LIN {X 0,Y 251.321,Z 689.744,A -85,B 0,C 180,E1 12849.752,E2 12849.752} C_VEL
LIN {X 0,Y 252.942,Z 676.86,A -85,B 0,C 180,E1 12846.595,E2 12846.595} C_VEL
LIN {X 0,Y 255.041,Z 662.352,A -85,B 0,C 180,E1 12843.706,E2 12843.706} C_VEL
LIN {X 0,Y 257.379,Z 646.816,A -85,B 0,C 180,E1 12841.205,E2 12841.205} C_VEL
LIN {X 0,Y 259.787,Z 630.262,A -85,B 0,C 180,E1 12839.084,E2 12839.084} C_VEL
LIN {X 0,Y 262.1,Z 612.775,A -85,B 0,C 180,E1 12837.333,E2 12837.333} C_VEL
LIN {X 0,Y 264.21,Z 594.401,A -85,B 0,C 180,E1 12835.941,E2 12835.941} C_VEL
LIN {X 0,Y 265.742,Z 575.64,A -85,B 0,C 180,E1 12834.93,E2 12834.93} C_VEL
LIN {X 0,Y 274.022,Z 424.566,A -85,B 0,C 180,E1 12829.575,E2 12829.575} C_VEL
LIN {X 0,Y 272.391,Z 392.722,A -85,B 0,C 180,E1 12828.155,E2 12828.155} C_VEL
LIN {X 0,Y 272.465,Z 390.527,A -85,B 0,C 180,E1 12828.028,E2 12828.028} C_VEL
LIN {X 0,Y 273.095,Z 387.473,A -85,B 0,C 180,E1 12827.542,E2 12827.542} C_VEL
LIN {X 0,Y 266.657,Z 366.923,A -85,B 0,C 180,E1 12823.018,E2 12823.018} C_VEL
LIN {X 0,Y 260.852,Z 349.171,A -85,B 0,C 180,E1 12818.67,E2 12818.67} C_VEL
LIN {X 0,Y 255.343,Z 333.14,A -85,B 0,C 180,E1 12814.327,E2 12814.327} C_VEL
LIN {X 0,Y 250.605,Z 319.583,A -85,B 0,C 180,E1 12810.252,E2 12810.252} C_VEL
LIN {X 0,Y 250.621,Z 319.582,A -85,B 0,C 180,E1 12805.526,E2 12805.526} C_VEL
LIN {X 0,Y 250.603,Z 319.579,A -85,B 0,C 180,E1 12800.558,E2 12800.558} C_VEL
LIN {X 0,Y 250.63,Z 319.58,A -85,B 0,C 180,E1 12795.506,E2 12795.506} C_VEL
LIN {X 0,Y 250.608,Z 319.58,A -85,B 0,C 180,E1 12790.346,E2 12790.346} C_VEL
LIN {X 0,Y 250.626,Z 319.579,A -85,B 0,C 180,E1 12785.497,E2 12785.497} C_VEL
LIN {X 0,Y 250.606,Z 319.58,A -85,B 0,C 180,E1 12780.46,E2 12780.46} C_VEL
LIN {X 0,Y 250.625,Z 319.576,A -85,B 0,C 180,E1 12775.427,E2 12775.427} C_VEL
LIN {X 0,Y 250.607,Z 319.572,A -85,B 0,C 180,E1 12770.589,E2 12770.589} C_VEL
LIN {X 0,Y 250.645,Z 319.578,A -85,B 0,C 180,E1 12765.448,E2 12765.448} C_VEL
LIN {X 0,Y 250.613,Z 319.565,A -85,B 0,C 180,E1 12760.309,E2 12760.309} C_VEL
LIN {X 0,Y 250.635,Z 319.578,A -85,B 0,C 180,E1 12755.44,E2 12755.44} C_VEL
LIN {X 0,Y 250.614,Z 319.559,A -85,B 0,C 180,E1 12750.425,E2 12750.425} C_VEL
LIN {X 0,Y 250.636,Z 319.579,A -85,B 0,C 180,E1 12745.5,E2 12745.5} C_VEL
LIN {X 0,Y 250.619,Z 319.565,A -85,B 0,C 180,E1 12740.634,E2 12740.634} C_VEL
LIN {X 0,Y 250.636,Z 319.572,A -85,B 0,C 180,E1 12735.565,E2 12735.565} C_VEL
LIN {X 0,Y 250.619,Z 319.573,A -85,B 0,C 180,E1 12730.562,E2 12730.562} C_VEL
LIN {X 0,Y 250.633,Z 319.56,A -85,B 0,C 180,E1 12725.536,E2 12725.536} C_VEL
LIN {X 0,Y 250.627,Z 319.577,A -85,B 0,C 180,E1 12720.705,E2 12720.705} C_VEL
LIN {X 0,Y 250.636,Z 319.561,A -85,B 0,C 180,E1 12715.644,E2 12715.644} C_VEL
LIN {X 0,Y 250.634,Z 319.574,A -85,B 0,C 180,E1 12710.794,E2 12710.794} C_VEL
LIN {X 0,Y 250.635,Z 319.571,A -85,B 0,C 180,E1 12705.738,E2 12705.738} C_VEL
LIN {X 0,Y 250.635,Z 319.574,A -85,B 0,C 180,E1 12700.805,E2 12700.805} C_VEL
LIN {X 0,Y 250.634,Z 319.573,A -85,B 0,C 180,E1 12695.722,E2 12695.722} C_VEL
LIN {X 0,Y 250.638,Z 319.575,A -85,B 0,C 180,E1 12690.684,E2 12690.684} C_VEL
LIN {X 0,Y 250.636,Z 319.567,A -85,B 0,C 180,E1 12685.651,E2 12685.651} C_VEL
LIN {X 0,Y 250.645,Z 319.572,A -85,B 0,C 180,E1 12680.817,E2 12680.817} C_VEL
LIN {X 0,Y 250.639,Z 319.578,A -85,B 0,C 180,E1 12675.679,E2 12675.679} C_VEL
LIN {X 0,Y 250.651,Z 319.575,A -85,B 0,C 180,E1 12670.905,E2 12670.905} C_VEL
LIN {X 0,Y 250.639,Z 319.578,A -85,B 0,C 180,E1 12665.737,E2 12665.737} C_VEL
LIN {X 0,Y 250.66,Z 319.574,A -85,B 0,C 180,E1 12660.867,E2 12660.867} C_VEL
LIN {X 0,Y 250.639,Z 319.575,A -85,B 0,C 180,E1 12655.77,E2 12655.77} C_VEL
LIN {X 0,Y 250.691,Z 319.79,A -85,B 0,C 180,E1 12651.229,E2 12651.229} C_VEL
LIN {X 0,Y 255.331,Z 334.84,A -85,B 0,C 180,E1 12646.417,E2 12646.417} C_VEL
LIN {X 0,Y 259.574,Z 349.98,A -85,B 0,C 180,E1 12641.974,E2 12641.974} C_VEL
LIN {X 0,Y 263.572,Z 365.649,A -85,B 0,C 180,E1 12637.706,E2 12637.706} C_VEL
LIN {X 0,Y 265.522,Z 374.511,A -85,B 0,C 180,E1 12635.439,E2 12635.439} C_VEL
LIN {X 0,Y 260.741,Z 400.55,A -85,B 0,C 180,E1 12630.016,E2 12630.016} C_VEL
LIN {X 0,Y 264.226,Z 442.101,A -85,B 0,C 180,E1 12627.745,E2 12627.745} C_VEL
LIN {X 0,Y 258.452,Z 538.649,A -85,B 0,C 180,E1 12623.423,E2 12623.423} C_VEL
LIN {X 0,Y 257.316,Z 556.591,A -85,B 0,C 180,E1 12622.208,E2 12622.208} C_VEL
LIN {X 0,Y 256.049,Z 573.142,A -85,B 0,C 180,E1 12620.691,E2 12620.691} C_VEL
LIN {X 0,Y 254.557,Z 590.125,A -85,B 0,C 180,E1 12618.666,E2 12618.666} C_VEL
LIN {X 0,Y 253.14,Z 605.769,A -85,B 0,C 180,E1 12616.283,E2 12616.283} C_VEL
LIN {X 0,Y 251.879,Z 620.01,A -85,B 0,C 180,E1 12613.541,E2 12613.541} C_VEL
LIN {X 0,Y 250.936,Z 632.25,A -85,B 0,C 180,E1 12610.558,E2 12610.558} C_VEL
LIN {X 0,Y 250.407,Z 642.044,A -85,B 0,C 180,E1 12607.568,E2 12607.568} C_VEL
LIN {X 0,Y 250.249,Z 650.429,A -85,B 0,C 180,E1 12604.35,E2 12604.35} C_VEL
LIN {X 0,Y 250.336,Z 654.067,A -85,B 0,C 180,E1 12602.603,E2 12602.603} C_VEL
LIN {X 0,Y 249.534,Z 657.084,A -85,B 0,C 180,E1 12600.972,E2 12600.972} C_VEL
LIN {X 0,Y 245.629,Z 662.003,A -85,B 0,C 180,E1 12597.788,E2 12597.788} C_VEL
LIN {X 0,Y 244.226,Z 664.446,A -85,B 0,C 180,E1 12595.666,E2 12595.666} C_VEL
LIN {X 0,Y 244.363,Z 665.1,A -85,B 0,C 180,E1 12594.901,E2 12594.901} C_VEL
LIN {X 0,Y 246.382,Z 667.107,A -85,B 0,C 180,E1 12591.361,E2 12591.361} C_VEL
LIN {X 0,Y 249.308,Z 667.226,A -85,B 0,C 180,E1 12587.725,E2 12587.725} C_VEL
LIN {X 0,Y 253.145,Z 665.497,A -85,B 0,C 180,E1 12584.182,E2 12584.182} C_VEL
LIN {X 0,Y 257.872,Z 661.812,A -85,B 0,C 180,E1 12580.754,E2 12580.754} C_VEL
LIN {X 0,Y 263.52,Z 656.236,A -85,B 0,C 180,E1 12577.464,E2 12577.464} C_VEL
LIN {X 0,Y 270.049,Z 648.574,A -85,B 0,C 180,E1 12574.327,E2 12574.327} C_VEL
LIN {X 0,Y 276.967,Z 639.386,A -85,B 0,C 180,E1 12571.539,E2 12571.539} C_VEL
LIN {X 0,Y 284.686,Z 628.026,A -85,B 0,C 180,E1 12568.914,E2 12568.914} C_VEL
LIN {X 0,Y 292.903,Z 614.48,A -85,B 0,C 180,E1 12566.541,E2 12566.541} C_VEL
LIN {X 0,Y 300.548,Z 600.238,A -85,B 0,C 180,E1 12564.627,E2 12564.627} C_VEL
LIN {X 0,Y 307.744,Z 584.985,A -85,B 0,C 180,E1 12563.051,E2 12563.051} C_VEL
LIN {X 0,Y 314.232,Z 568.47,A -85,B 0,C 180,E1 12561.763,E2 12561.763} C_VEL
LIN {X 0,Y 319.672,Z 551.343,A -85,B 0,C 180,E1 12560.771,E2 12560.771} C_VEL
LIN {X 0,Y 325.594,Z 530.519,A -85,B 0,C 180,E1 12559.792,E2 12559.792} C_VEL
LIN {X 0,Y 315.19,Z 568.695,A -85,B 0,C 180,E1 12558.338,E2 12558.338} C_VEL
LIN {X 0,Y 307.601,Z 590.208,A -85,B 0,C 180,E1 12557.276,E2 12557.276} C_VEL
LIN {X 0,Y 299.978,Z 608.25,A -85,B 0,C 180,E1 12556.052,E2 12556.052} C_VEL
LIN {X 0,Y 291.443,Z 626.077,A -85,B 0,C 180,E1 12554.418,E2 12554.418} C_VEL
LIN {X 0,Y 282.982,Z 642.204,A -85,B 0,C 180,E1 12552.445,E2 12552.445} C_VEL
LIN {X 0,Y 274.169,Z 657.891,A -85,B 0,C 180,E1 12549.932,E2 12549.932} C_VEL
LIN {X 0,Y 265.896,Z 672.135,A -85,B 0,C 180,E1 12546.99,E2 12546.99} C_VEL
LIN {X 0,Y 258.373,Z 684.983,A -85,B 0,C 180,E1 12543.601,E2 12543.601} C_VEL
LIN {X 0,Y 251.862,Z 696.369,A -85,B 0,C 180,E1 12539.753,E2 12539.753} C_VEL
LIN {X 0,Y 246.671,Z 706.308,A -85,B 0,C 180,E1 12535.448,E2 12535.448} C_VEL
LIN {X 0,Y 243.156,Z 714.309,A -85,B 0,C 180,E1 12530.964,E2 12530.964} C_VEL
LIN {X 0,Y 241.284,Z 720.475,A -85,B 0,C 180,E1 12526.369,E2 12526.369} C_VEL
LIN {X 0,Y 240.873,Z 724.951,A -85,B 0,C 180,E1 12521.574,E2 12521.574} C_VEL
LIN {X 0,Y 241.603,Z 727.321,A -85,B 0,C 180,E1 12517.134,E2 12517.134} C_VEL
LIN {X 0,Y 242.656,Z 727.848,A -85,B 0,C 180,E1 12513.309,E2 12513.309} C_VEL
LIN {X 0,Y 243.307,Z 726.953,A -85,B 0,C 180,E1 12510.002,E2 12510.002} C_VEL
LIN {X 0,Y 243.197,Z 724.887,A -85,B 0,C 180,E1 12506.938,E2 12506.938} C_VEL
LIN {X 0,Y 242.612,Z 720.804,A -85,B 0,C 180,E1 12503.34,E2 12503.34} C_VEL
LIN {X 0,Y 242.105,Z 715.047,A -85,B 0,C 180,E1 12499.773,E2 12499.773} C_VEL
LIN {X 0,Y 242.009,Z 707.373,A -85,B 0,C 180,E1 12496.137,E2 12496.137} C_VEL
LIN {X 0,Y 242.521,Z 697.577,A -85,B 0,C 180,E1 12492.487,E2 12492.487} C_VEL
LIN {X 0,Y 243.672,Z 686.258,A -85,B 0,C 180,E1 12489.087,E2 12489.087} C_VEL
LIN {X 0,Y 245.402,Z 673.121,A -85,B 0,C 180,E1 12485.881,E2 12485.881} C_VEL
LIN {X 0,Y 247.487,Z 659.126,A -85,B 0,C 180,E1 12483.099,E2 12483.099} C_VEL
LIN {X 0,Y 249.818,Z 643.804,A -85,B 0,C 180,E1 12480.643,E2 12480.643} C_VEL
LIN {X 0,Y 252.319,Z 626.753,A -85,B 0,C 180,E1 12478.464,E2 12478.464} C_VEL
LIN {X 0,Y 254.732,Z 608.718,A -85,B 0,C 180,E1 12476.668,E2 12476.668} C_VEL
LIN {X 0,Y 256.805,Z 590.184,A -85,B 0,C 180,E1 12475.305,E2 12475.305} C_VEL
LIN {X 0,Y 258.241,Z 570.947,A -85,B 0,C 180,E1 12474.319,E2 12474.319} C_VEL
LIN {X 0,Y 266.563,Z 425.162,A -85,B 0,C 180,E1 12468.963,E2 12468.963} C_VEL
LIN {X 0,Y 265.03,Z 393.337,A -85,B 0,C 180,E1 12467.5,E2 12467.5} C_VEL
LIN {X 0,Y 265.123,Z 390.585,A -85,B 0,C 180,E1 12467.344,E2 12467.344} C_VEL
LIN {X 0,Y 265.183,Z 388.765,A -85,B 0,C 180,E1 12467.013,E2 12467.013} C_VEL
LIN {X 0,Y 258.711,Z 367.881,A -85,B 0,C 180,E1 12462.261,E2 12462.261} C_VEL
LIN {X 0,Y 252.668,Z 349.364,A -85,B 0,C 180,E1 12457.55,E2 12457.55} C_VEL
LIN {X 0,Y 246.993,Z 332.812,A -85,B 0,C 180,E1 12452.854,E2 12452.854} C_VEL
LIN {X 0,Y 242.667,Z 320.567,A -85,B 0,C 180,E1 12448.963,E2 12448.963} C_VEL
LIN {X 0,Y 242.684,Z 320.567,A -85,B 0,C 180,E1 12443.817,E2 12443.817} C_VEL
LIN {X 0,Y 242.666,Z 320.572,A -85,B 0,C 180,E1 12438.75,E2 12438.75} C_VEL
LIN {X 0,Y 242.686,Z 320.564,A -85,B 0,C 180,E1 12433.828,E2 12433.828} C_VEL
LIN {X 0,Y 242.665,Z 320.562,A -85,B 0,C 180,E1 12428.772,E2 12428.772} C_VEL
LIN {X 0,Y 242.681,Z 320.563,A -85,B 0,C 180,E1 12423.783,E2 12423.783} C_VEL
LIN {X 0,Y 242.671,Z 320.566,A -85,B 0,C 180,E1 12418.823,E2 12418.823} C_VEL
LIN {X 0,Y 242.696,Z 320.569,A -85,B 0,C 180,E1 12413.617,E2 12413.617} C_VEL
LIN {X 0,Y 242.671,Z 320.561,A -85,B 0,C 180,E1 12408.597,E2 12408.597} C_VEL
LIN {X 0,Y 242.695,Z 320.563,A -85,B 0,C 180,E1 12403.489,E2 12403.489} C_VEL
LIN {X 0,Y 242.676,Z 320.563,A -85,B 0,C 180,E1 12398.492,E2 12398.492} C_VEL
LIN {X 0,Y 242.698,Z 320.559,A -85,B 0,C 180,E1 12393.374,E2 12393.374} C_VEL
LIN {X 0,Y 242.678,Z 320.558,A -85,B 0,C 180,E1 12388.454,E2 12388.454} C_VEL
LIN {X 0,Y 242.696,Z 320.564,A -85,B 0,C 180,E1 12383.449,E2 12383.449} C_VEL
LIN {X 0,Y 242.679,Z 320.547,A -85,B 0,C 180,E1 12378.451,E2 12378.451} C_VEL
LIN {X 0,Y 242.7,Z 320.567,A -85,B 0,C 180,E1 12373.469,E2 12373.469} C_VEL
LIN {X 0,Y 242.681,Z 320.553,A -85,B 0,C 180,E1 12368.469,E2 12368.469} C_VEL
LIN {X 0,Y 242.702,Z 320.561,A -85,B 0,C 180,E1 12363.257,E2 12363.257} C_VEL
LIN {X 0,Y 242.688,Z 320.563,A -85,B 0,C 180,E1 12358.166,E2 12358.166} C_VEL
LIN {X 0,Y 242.703,Z 320.552,A -85,B 0,C 180,E1 12353.038,E2 12353.038} C_VEL
LIN {X 0,Y 242.696,Z 320.566,A -85,B 0,C 180,E1 12347.748,E2 12347.748} C_VEL
LIN {X 0,Y 242.698,Z 320.552,A -85,B 0,C 180,E1 12342.852,E2 12342.852} C_VEL
LIN {X 0,Y 242.702,Z 320.567,A -85,B 0,C 180,E1 12337.574,E2 12337.574} C_VEL
LIN {X 0,Y 242.693,Z 320.559,A -85,B 0,C 180,E1 12332.596,E2 12332.596} C_VEL
LIN {X 0,Y 242.704,Z 320.559,A -85,B 0,C 180,E1 12327.401,E2 12327.401} C_VEL
LIN {X 0,Y 242.694,Z 320.565,A -85,B 0,C 180,E1 12322.423,E2 12322.423} C_VEL
LIN {X 0,Y 242.708,Z 320.564,A -85,B 0,C 180,E1 12317.387,E2 12317.387} C_VEL
LIN {X 0,Y 242.7,Z 320.563,A -85,B 0,C 180,E1 12312.496,E2 12312.496} C_VEL
LIN {X 0,Y 242.724,Z 320.566,A -85,B 0,C 180,E1 12307.217,E2 12307.217} C_VEL
LIN {X 0,Y 242.701,Z 320.567,A -85,B 0,C 180,E1 12302.254,E2 12302.254} C_VEL
LIN {X 0,Y 242.718,Z 320.564,A -85,B 0,C 180,E1 12297.17,E2 12297.17} C_VEL
LIN {X 0,Y 242.708,Z 320.589,A -85,B 0,C 180,E1 12292.43,E2 12292.43} C_VEL
LIN {X 0,Y 247.265,Z 335.339,A -85,B 0,C 180,E1 12287.521,E2 12287.521} C_VEL
LIN {X 0,Y 251.505,Z 350.2,A -85,B 0,C 180,E1 12282.986,E2 12282.986} C_VEL
LIN {X 0,Y 255.595,Z 366.284,A -85,B 0,C 180,E1 12278.456,E2 12278.456} C_VEL
LIN {X 0,Y 257.838,Z 376.167,A -85,B 0,C 180,E1 12275.837,E2 12275.837} C_VEL
LIN {X 0,Y 253.208,Z 400.564,A -85,B 0,C 180,E1 12270.66,E2 12270.66} C_VEL
LIN {X 0,Y 256.409,Z 441.043,A -85,B 0,C 180,E1 12268.368,E2 12268.368} C_VEL
LIN {X 0,Y 256.416,Z 446.756,A -85,B 0,C 180,E1 12268.085,E2 12268.085} C_VEL
LIN {X 0,Y 250.616,Z 539.133,A -85,B 0,C 180,E1 12263.788,E2 12263.788} C_VEL
LIN {X 0,Y 249.42,Z 557.457,A -85,B 0,C 180,E1 12262.505,E2 12262.505} C_VEL
LIN {X 0,Y 248.079,Z 574.425,A -85,B 0,C 180,E1 12260.893,E2 12260.893} C_VEL
LIN {X 0,Y 246.636,Z 590.499,A -85,B 0,C 180,E1 12258.92,E2 12258.92} C_VEL
LIN {X 0,Y 245.114,Z 606.831,A -85,B 0,C 180,E1 12256.344,E2 12256.344} C_VEL
LIN {X 0,Y 243.838,Z 621.036,A -85,B 0,C 180,E1 12253.513,E2 12253.513} C_VEL
LIN {X 0,Y 242.86,Z 633.967,A -85,B 0,C 180,E1 12250.265,E2 12250.265} C_VEL
LIN {X 0,Y 242.364,Z 643.889,A -85,B 0,C 180,E1 12247.106,E2 12247.106} C_VEL
LIN {X 0,Y 242.273,Z 652.096,A -85,B 0,C 180,E1 12243.783,E2 12243.783} C_VEL
LIN {X 0,Y 242.676,Z 658.769,A -85,B 0,C 180,E1 12240.233,E2 12240.233} C_VEL
LIN {X 0,Y 243.628,Z 663.41,A -85,B 0,C 180,E1 12236.703,E2 12236.703} C_VEL
LIN {X 0,Y 244.363,Z 665.1,A -85,B 0,C 180,E1 12234.901,E2 12234.901} C_VEL
LIN {X 0,Y 244.306,Z 666.547,A -85,B 0,C 180,E1 12233.11,E2 12233.11} C_VEL
LIN {X 0,Y 241.997,Z 668.588,A -85,B 0,C 180,E1 12229.49,E2 12229.49} C_VEL
LIN {X 0,Y 241.842,Z 668.966,A -85,B 0,C 180,E1 12227.384,E2 12227.384} C_VEL
LIN {X 0,Y 242.405,Z 668.865,A -85,B 0,C 180,E1 12226.608,E2 12226.608} C_VEL
LIN {X 0,Y 246.611,Z 667.235,A -85,B 0,C 180,E1 12223.024,E2 12223.024} C_VEL
LIN {X 0,Y 252.134,Z 663.404,A -85,B 0,C 180,E1 12219.33,E2 12219.33} C_VEL
LIN {X 0,Y 258.313,Z 657.897,A -85,B 0,C 180,E1 12216.017,E2 12216.017} C_VEL
LIN {X 0,Y 265.885,Z 649.875,A -85,B 0,C 180,E1 12212.689,E2 12212.689} C_VEL
LIN {X 0,Y 273.919,Z 640.089,A -85,B 0,C 180,E1 12209.75,E2 12209.75} C_VEL
LIN {X 0,Y 281.716,Z 629.576,A -85,B 0,C 180,E1 12207.349,E2 12207.349} C_VEL
LIN {X 0,Y 290.837,Z 615.795,A -85,B 0,C 180,E1 12204.959,E2 12204.959} C_VEL
LIN {X 0,Y 299.337,Z 601.152,A -85,B 0,C 180,E1 12203.038,E2 12203.038} C_VEL
LIN {X 0,Y 306.983,Z 586.005,A -85,B 0,C 180,E1 12201.528,E2 12201.528} C_VEL
LIN {X 0,Y 313.846,Z 569.643,A -85,B 0,C 180,E1 12200.298,E2 12200.298} C_VEL
LIN {X 0,Y 315.67,Z 564.662,A -85,B 0,C 180,E1 12199.974,E2 12199.974} C_VEL
LIN {X 0,Y 308.363,Z 584.784,A -85,B 0,C 180,E1 12199.071,E2 12199.071} C_VEL
LIN {X 0,Y 300.287,Z 603.247,A -85,B 0,C 180,E1 12197.948,E2 12197.948} C_VEL
LIN {X 0,Y 291.905,Z 619.971,A -85,B 0,C 180,E1 12196.567,E2 12196.567} C_VEL
LIN {X 0,Y 282.694,Z 636.496,A -85,B 0,C 180,E1 12194.738,E2 12194.738} C_VEL
LIN {X 0,Y 273.343,Z 652.123,A -85,B 0,C 180,E1 12192.447,E2 12192.447} C_VEL
LIN {X 0,Y 264.372,Z 666.297,A -85,B 0,C 180,E1 12189.731,E2 12189.731} C_VEL
LIN {X 0,Y 255.765,Z 679.533,A -85,B 0,C 180,E1 12186.458,E2 12186.458} C_VEL
LIN {X 0,Y 248.108,Z 691.408,A -85,B 0,C 180,E1 12182.686,E2 12182.686} C_VEL
LIN {X 0,Y 241.723,Z 701.854,A -85,B 0,C 180,E1 12178.406,E2 12178.406} C_VEL
LIN {X 0,Y 236.899,Z 710.699,A -85,B 0,C 180,E1 12173.64,E2 12173.64} C_VEL
LIN {X 0,Y 233.993,Z 717.563,A -85,B 0,C 180,E1 12168.694,E2 12168.694} C_VEL
LIN {X 0,Y 232.915,Z 722.497,A -85,B 0,C 180,E1 12163.659,E2 12163.659} C_VEL
LIN {X 0,Y 233.302,Z 725.357,A -85,B 0,C 180,E1 12158.877,E2 12158.877} C_VEL
LIN {X 0,Y 234.403,Z 726.281,A -85,B 0,C 180,E1 12154.651,E2 12154.651} C_VEL
LIN {X 0,Y 235.306,Z 725.756,A -85,B 0,C 180,E1 12151.219,E2 12151.219} C_VEL
LIN {X 0,Y 235.505,Z 724.163,A -85,B 0,C 180,E1 12148.299,E2 12148.299} C_VEL
LIN {X 0,Y 235.057,Z 720.878,A -85,B 0,C 180,E1 12144.877,E2 12144.877} C_VEL
LIN {X 0,Y 234.432,Z 715.636,A -85,B 0,C 180,E1 12141.17,E2 12141.17} C_VEL
LIN {X 0,Y 234.132,Z 708.006,A -85,B 0,C 180,E1 12137.172,E2 12137.172} C_VEL
LIN {X 0,Y 234.446,Z 698.755,A -85,B 0,C 180,E1 12133.399,E2 12133.399} C_VEL
LIN {X 0,Y 235.444,Z 687.784,A -85,B 0,C 180,E1 12129.811,E2 12129.811} C_VEL
LIN {X 0,Y 237.101,Z 674.719,A -85,B 0,C 180,E1 12126.385,E2 12126.385} C_VEL
LIN {X 0,Y 239.257,Z 660.214,A -85,B 0,C 180,E1 12123.307,E2 12123.307} C_VEL
LIN {X 0,Y 241.672,Z 644.673,A -85,B 0,C 180,E1 12120.644,E2 12120.644} C_VEL
LIN {X 0,Y 244.173,Z 628.063,A -85,B 0,C 180,E1 12118.392,E2 12118.392} C_VEL
LIN {X 0,Y 246.748,Z 609.361,A -85,B 0,C 180,E1 12116.421,E2 12116.421} C_VEL
LIN {X 0,Y 248.816,Z 591.743,A -85,B 0,C 180,E1 12115.026,E2 12115.026} C_VEL
LIN {X 0,Y 250.347,Z 572.991,A -85,B 0,C 180,E1 12113.98,E2 12113.98} C_VEL
LIN {X 0,Y 259.11,Z 425.76,A -85,B 0,C 180,E1 12108.332,E2 12108.332} C_VEL
LIN {X 0,Y 257.668,Z 393.859,A -85,B 0,C 180,E1 12106.822,E2 12106.822} C_VEL
LIN {X 0,Y 257.53,Z 390.861,A -85,B 0,C 180,E1 12106.638,E2 12106.638} C_VEL
LIN {X 0,Y 251.329,Z 370.698,A -85,B 0,C 180,E1 12101.935,E2 12101.935} C_VEL
LIN {X 0,Y 245.628,Z 353.059,A -85,B 0,C 180,E1 12097.342,E2 12097.342} C_VEL
LIN {X 0,Y 239.968,Z 336.421,A -85,B 0,C 180,E1 12092.517,E2 12092.517} C_VEL
LIN {X 0,Y 235.324,Z 323.746,A -85,B 0,C 180,E1 12088.419,E2 12088.419} C_VEL
LIN {X 0,Y 234.751,Z 321.557,A -85,B 0,C 180,E1 12087.64,E2 12087.64} C_VEL
LIN {X 0,Y 234.73,Z 321.562,A -85,B 0,C 180,E1 12082.281,E2 12082.281} C_VEL
LIN {X 0,Y 234.74,Z 321.553,A -85,B 0,C 180,E1 12077.35,E2 12077.35} C_VEL
LIN {X 0,Y 234.734,Z 321.555,A -85,B 0,C 180,E1 12072.05,E2 12072.05} C_VEL
LIN {X 0,Y 234.735,Z 321.559,A -85,B 0,C 180,E1 12067.053,E2 12067.053} C_VEL
LIN {X 0,Y 234.748,Z 321.554,A -85,B 0,C 180,E1 12061.712,E2 12061.712} C_VEL
LIN {X 0,Y 234.73,Z 321.548,A -85,B 0,C 180,E1 12056.585,E2 12056.585} C_VEL
LIN {X 0,Y 234.755,Z 321.549,A -85,B 0,C 180,E1 12051.431,E2 12051.431} C_VEL
LIN {X 0,Y 234.737,Z 321.557,A -85,B 0,C 180,E1 12046.198,E2 12046.198} C_VEL
LIN {X 0,Y 234.745,Z 321.54,A -85,B 0,C 180,E1 12041.117,E2 12041.117} C_VEL
LIN {X 0,Y 234.747,Z 321.557,A -85,B 0,C 180,E1 12035.869,E2 12035.869} C_VEL
LIN {X 0,Y 234.741,Z 321.534,A -85,B 0,C 180,E1 12030.826,E2 12030.826} C_VEL
LIN {X 0,Y 234.758,Z 321.556,A -85,B 0,C 180,E1 12025.501,E2 12025.501} C_VEL
LIN {X 0,Y 234.739,Z 321.541,A -85,B 0,C 180,E1 12020.294,E2 12020.294} C_VEL
LIN {X 0,Y 234.759,Z 321.55,A -85,B 0,C 180,E1 12015.335,E2 12015.335} C_VEL
LIN {X 0,Y 234.746,Z 321.551,A -85,B 0,C 180,E1 12010.025,E2 12010.025} C_VEL
LIN {X 0,Y 234.757,Z 321.539,A -85,B 0,C 180,E1 12005.096,E2 12005.096} C_VEL
LIN {X 0,Y 234.754,Z 321.555,A -85,B 0,C 180,E1 11999.887,E2 11999.887} C_VEL
LIN {X 0,Y 234.755,Z 321.531,A -85,B 0,C 180,E1 11994.89,E2 11994.89} C_VEL
LIN {X 0,Y 234.76,Z 321.554,A -85,B 0,C 180,E1 11989.66,E2 11989.66} C_VEL
LIN {X 0,Y 234.747,Z 321.541,A -85,B 0,C 180,E1 11984.552,E2 11984.552} C_VEL
LIN {X 0,Y 234.767,Z 321.556,A -85,B 0,C 180,E1 11979.312,E2 11979.312} C_VEL
LIN {X 0,Y 234.747,Z 321.542,A -85,B 0,C 180,E1 11974.395,E2 11974.395} C_VEL
LIN {X 0,Y 234.778,Z 321.553,A -85,B 0,C 180,E1 11969.266,E2 11969.266} C_VEL
LIN {X 0,Y 234.756,Z 321.551,A -85,B 0,C 180,E1 11963.886,E2 11963.886} C_VEL
LIN {X 0,Y 234.766,Z 321.546,A -85,B 0,C 180,E1 11958.949,E2 11958.949} C_VEL
LIN {X 0,Y 234.761,Z 321.548,A -85,B 0,C 180,E1 11953.672,E2 11953.672} C_VEL
LIN {X 0,Y 234.77,Z 321.549,A -85,B 0,C 180,E1 11948.775,E2 11948.775} C_VEL
LIN {X 0,Y 234.773,Z 321.556,A -85,B 0,C 180,E1 11943.415,E2 11943.415} C_VEL
LIN {X 0,Y 234.765,Z 321.551,A -85,B 0,C 180,E1 11938.399,E2 11938.399} C_VEL
LIN {X 0,Y 234.787,Z 321.701,A -85,B 0,C 180,E1 11933.59,E2 11933.59} C_VEL
LIN {X 0,Y 239.057,Z 335.38,A -85,B 0,C 180,E1 11928.831,E2 11928.831} C_VEL
LIN {X 0,Y 243.141,Z 349.561,A -85,B 0,C 180,E1 11924.311,E2 11924.311} C_VEL
LIN {X 0,Y 247.162,Z 365.017,A -85,B 0,C 180,E1 11919.768,E2 11919.768} C_VEL
LIN {X 0,Y 250.141,Z 377.771,A -85,B 0,C 180,E1 11916.264,E2 11916.264} C_VEL
LIN {X 0,Y 245.67,Z 400.359,A -85,B 0,C 180,E1 11911.33,E2 11911.33} C_VEL
LIN {X 0,Y 248.522,Z 439.066,A -85,B 0,C 180,E1 11909.065,E2 11909.065} C_VEL
LIN {X 0,Y 248.874,Z 445.916,A -85,B 0,C 180,E1 11908.687,E2 11908.687} C_VEL
LIN {X 0,Y 242.779,Z 539.749,A -85,B 0,C 180,E1 11904.162,E2 11904.162} C_VEL
LIN {X 0,Y 241.539,Z 558.007,A -85,B 0,C 180,E1 11902.831,E2 11902.831} C_VEL
LIN {X 0,Y 240.079,Z 575.771,A -85,B 0,C 180,E1 11901.066,E2 11901.066} C_VEL
LIN {X 0,Y 238.562,Z 592.199,A -85,B 0,C 180,E1 11898.95,E2 11898.95} C_VEL
LIN {X 0,Y 237.088,Z 607.78,A -85,B 0,C 180,E1 11896.409,E2 11896.409} C_VEL
LIN {X 0,Y 235.797,Z 622.061,A -85,B 0,C 180,E1 11893.483,E2 11893.483} C_VEL
LIN {X 0,Y 234.899,Z 633.699,A -85,B 0,C 180,E1 11890.49,E2 11890.49} C_VEL
LIN {X 0,Y 234.388,Z 643.586,A -85,B 0,C 180,E1 11887.349,E2 11887.349} C_VEL
LIN {X 0,Y 234.277,Z 652.202,A -85,B 0,C 180,E1 11883.912,E2 11883.912} C_VEL
LIN {X 0,Y 234.64,Z 658.79,A -85,B 0,C 180,E1 11880.485,E2 11880.485} C_VEL
LIN {X 0,Y 235.685,Z 664.241,A -85,B 0,C 180,E1 11876.592,E2 11876.592} C_VEL
LIN {X 0,Y 237.37,Z 667.418,A -85,B 0,C 180,E1 11872.98,E2 11872.98} C_VEL
LIN {X 0,Y 240.021,Z 668.959,A -85,B 0,C 180,E1 11869.192,E2 11869.192} C_VEL
LIN {X 0,Y 242.405,Z 668.865,A -85,B 0,C 180,E1 11866.608,E2 11866.608} C_VEL
LIN {X 0,Y 243.444,Z 668.608,A -85,B 0,C 180,E1 11864.659,E2 11864.659} C_VEL
LIN {X 0,Y 243.672,Z 667.527,A -85,B 0,C 180,E1 11860.46,E2 11860.46} C_VEL
LIN {X 0,Y 245.139,Z 666.156,A -85,B 0,C 180,E1 11858.709,E2 11858.709} C_VEL
LIN {X 0,Y 245.696,Z 665.742,A -85,B 0,C 180,E1 11858.357,E2 11858.357} C_VEL
LIN {X 0,Y 252.46,Z 660.483,A -85,B 0,C 180,E1 11854.924,E2 11854.924} C_VEL
LIN {X 0,Y 260.005,Z 653.391,A -85,B 0,C 180,E1 11851.768,E2 11851.768} C_VEL
LIN {X 0,Y 268.479,Z 644.341,A -85,B 0,C 180,E1 11848.822,E2 11848.822} C_VEL
LIN {X 0,Y 277.857,Z 632.992,A -85,B 0,C 180,E1 11846.096,E2 11846.096} C_VEL
LIN {X 0,Y 286.812,Z 620.84,A -85,B 0,C 180,E1 11843.901,E2 11843.901} C_VEL
LIN {X 0,Y 296.067,Z 606.682,A -85,B 0,C 180,E1 11841.949,E2 11841.949} C_VEL
LIN {X 0,Y 304.755,Z 591.155,A -85,B 0,C 180,E1 11840.345,E2 11840.345} C_VEL
LIN {X 0,Y 304.991,Z 590.733,A -85,B 0,C 180,E1 11840.276,E2 11840.276} C_VEL
LIN {X 0,Y 295.819,Z 609.276,A -85,B 0,C 180,E1 11839.064,E2 11839.064} C_VEL
LIN {X 0,Y 286.089,Z 626.39,A -85,B 0,C 180,E1 11837.515,E2 11837.515} C_VEL
LIN {X 0,Y 276.017,Z 642.495,A -85,B 0,C 180,E1 11835.532,E2 11835.532} C_VEL
LIN {X 0,Y 266.181,Z 657.174,A -85,B 0,C 180,E1 11833.131,E2 11833.131} C_VEL
LIN {X 0,Y 256.747,Z 670.531,A -85,B 0,C 180,E1 11830.277,E2 11830.277} C_VEL
LIN {X 0,Y 247.512,Z 683.335,A -85,B 0,C 180,E1 11826.719,E2 11826.719} C_VEL
LIN {X 0,Y 239.41,Z 694.715,A -85,B 0,C 180,E1 11822.6,E2 11822.6} C_VEL
LIN {X 0,Y 233.108,Z 704.115,A -85,B 0,C 180,E1 11818.154,E2 11818.154} C_VEL
LIN {X 0,Y 228.403,Z 712.061,A -85,B 0,C 180,E1 11813.171,E2 11813.171} C_VEL
LIN {X 0,Y 225.747,Z 718.044,A -85,B 0,C 180,E1 11808.063,E2 11808.063} C_VEL
LIN {X 0,Y 224.942,Z 722.191,A -85,B 0,C 180,E1 11802.843,E2 11802.843} C_VEL
LIN {X 0,Y 225.616,Z 724.333,A -85,B 0,C 180,E1 11797.898,E2 11797.898} C_VEL
LIN {X 0,Y 226.892,Z 724.594,A -85,B 0,C 180,E1 11793.539,E2 11793.539} C_VEL
LIN {X 0,Y 227.66,Z 723.593,A -85,B 0,C 180,E1 11790.254,E2 11790.254} C_VEL
LIN {X 0,Y 227.592,Z 721.201,A -85,B 0,C 180,E1 11786.98,E2 11786.98} C_VEL
LIN {X 0,Y 226.977,Z 717.112,A -85,B 0,C 180,E1 11783.425,E2 11783.425} C_VEL
LIN {X 0,Y 226.405,Z 710.967,A -85,B 0,C 180,E1 11779.57,E2 11779.57} C_VEL
LIN {X 0,Y 226.321,Z 702.882,A -85,B 0,C 180,E1 11775.678,E2 11775.678} C_VEL
LIN {X 0,Y 226.865,Z 693.375,A -85,B 0,C 180,E1 11772.033,E2 11772.033} C_VEL
LIN {X 0,Y 228.11,Z 681.678,A -85,B 0,C 180,E1 11768.398,E2 11768.398} C_VEL
LIN {X 0,Y 229.948,Z 668.308,A -85,B 0,C 180,E1 11765.055,E2 11765.055} C_VEL
LIN {X 0,Y 232.278,Z 653.272,A -85,B 0,C 180,E1 11762.02,E2 11762.02} C_VEL
LIN {X 0,Y 234.808,Z 637.208,A -85,B 0,C 180,E1 11759.415,E2 11759.415} C_VEL
LIN {X 0,Y 237.359,Z 620.07,A -85,B 0,C 180,E1 11757.23,E2 11757.23} C_VEL
LIN {X 0,Y 239.773,Z 601.881,A -85,B 0,C 180,E1 11755.453,E2 11755.453} C_VEL
LIN {X 0,Y 241.821,Z 582.924,A -85,B 0,C 180,E1 11754.089,E2 11754.089} C_VEL
LIN {X 0,Y 243.183,Z 562.214,A -85,B 0,C 180,E1 11753.094,E2 11753.094} C_VEL
LIN {X 0,Y 251.641,Z 426.397,A -85,B 0,C 180,E1 11747.696,E2 11747.696} C_VEL
LIN {X 0,Y 250.302,Z 394.558,A -85,B 0,C 180,E1 11746.136,E2 11746.136} C_VEL
LIN {X 0,Y 249.628,Z 391.999,A -85,B 0,C 180,E1 11745.952,E2 11745.952} C_VEL
LIN {X 0,Y 249.012,Z 390.099,A -85,B 0,C 180,E1 11745.624,E2 11745.624} C_VEL
LIN {X 0,Y 243.152,Z 371.087,A -85,B 0,C 180,E1 11740.989,E2 11740.989} C_VEL
LIN {X 0,Y 237.69,Z 354.076,A -85,B 0,C 180,E1 11736.382,E2 11736.382} C_VEL
LIN {X 0,Y 232.368,Z 338.417,A -85,B 0,C 180,E1 11731.669,E2 11731.669} C_VEL
LIN {X 0,Y 227.559,Z 325.099,A -85,B 0,C 180,E1 11727.194,E2 11727.194} C_VEL
LIN {X 0,Y 226.791,Z 322.545,A -85,B 0,C 180,E1 11726.302,E2 11726.302} C_VEL
LIN {X 0,Y 226.798,Z 322.546,A -85,B 0,C 180,E1 11721.196,E2 11721.196} C_VEL
LIN {X 0,Y 226.807,Z 322.544,A -85,B 0,C 180,E1 11715.865,E2 11715.865} C_VEL
LIN {X 0,Y 226.79,Z 322.547,A -85,B 0,C 180,E1 11710.674,E2 11710.674} C_VEL
LIN {X 0,Y 226.809,Z 322.547,A -85,B 0,C 180,E1 11705.569,E2 11705.569} C_VEL
LIN {X 0,Y 226.793,Z 322.547,A -85,B 0,C 180,E1 11700.256,E2 11700.256} C_VEL
LIN {X 0,Y 226.799,Z 322.545,A -85,B 0,C 180,E1 11695.067,E2 11695.067} C_VEL
LIN {X 0,Y 226.803,Z 322.533,A -85,B 0,C 180,E1 11689.847,E2 11689.847} C_VEL
LIN {X 0,Y 226.797,Z 322.546,A -85,B 0,C 180,E1 11684.666,E2 11684.666} C_VEL
LIN {X 0,Y 226.816,Z 322.533,A -85,B 0,C 180,E1 11679.354,E2 11679.354} C_VEL
LIN {X 0,Y 226.804,Z 322.544,A -85,B 0,C 180,E1 11674.065,E2 11674.065} C_VEL
LIN {X 0,Y 226.811,Z 322.531,A -85,B 0,C 180,E1 11668.956,E2 11668.956} C_VEL
LIN {X 0,Y 226.812,Z 322.545,A -85,B 0,C 180,E1 11663.773,E2 11663.773} C_VEL
LIN {X 0,Y 226.802,Z 322.521,A -85,B 0,C 180,E1 11658.609,E2 11658.609} C_VEL
LIN {X 0,Y 226.82,Z 322.544,A -85,B 0,C 180,E1 11653.342,E2 11653.342} C_VEL
LIN {X 0,Y 226.805,Z 322.526,A -85,B 0,C 180,E1 11648.108,E2 11648.108} C_VEL
LIN {X 0,Y 226.816,Z 322.54,A -85,B 0,C 180,E1 11642.832,E2 11642.832} C_VEL
LIN {X 0,Y 226.825,Z 322.535,A -85,B 0,C 180,E1 11637.569,E2 11637.569} C_VEL
LIN {X 0,Y 226.806,Z 322.534,A -85,B 0,C 180,E1 11632.228,E2 11632.228} C_VEL
LIN {X 0,Y 226.826,Z 322.539,A -85,B 0,C 180,E1 11627.176,E2 11627.176} C_VEL
LIN {X 0,Y 226.812,Z 322.532,A -85,B 0,C 180,E1 11621.886,E2 11621.886} C_VEL
LIN {X 0,Y 226.824,Z 322.54,A -85,B 0,C 180,E1 11616.833,E2 11616.833} C_VEL
LIN {X 0,Y 226.825,Z 322.539,A -85,B 0,C 180,E1 11611.514,E2 11611.514} C_VEL
LIN {X 0,Y 226.814,Z 322.532,A -85,B 0,C 180,E1 11606.46,E2 11606.46} C_VEL
LIN {X 0,Y 226.831,Z 322.541,A -85,B 0,C 180,E1 11601.379,E2 11601.379} C_VEL
LIN {X 0,Y 226.815,Z 322.544,A -85,B 0,C 180,E1 11596.227,E2 11596.227} C_VEL
LIN {X 0,Y 226.835,Z 322.542,A -85,B 0,C 180,E1 11590.961,E2 11590.961} C_VEL
LIN {X 0,Y 226.828,Z 322.541,A -85,B 0,C 180,E1 11585.519,E2 11585.519} C_VEL
LIN {X 0,Y 226.824,Z 322.544,A -85,B 0,C 180,E1 11580.414,E2 11580.414} C_VEL
LIN {X 0,Y 226.833,Z 322.54,A -85,B 0,C 180,E1 11575.064,E2 11575.064} C_VEL
LIN {X 0,Y 226.904,Z 323.013,A -85,B 0,C 180,E1 11574.74,E2 11574.74} C_VEL
LIN {X 0,Y 231.083,Z 336.115,A -85,B 0,C 180,E1 11569.976,E2 11569.976} C_VEL
LIN {X 0,Y 235.242,Z 350.468,A -85,B 0,C 180,E1 11565.213,E2 11565.213} C_VEL
LIN {X 0,Y 239.269,Z 366.014,A -85,B 0,C 180,E1 11560.485,E2 11560.485} C_VEL
LIN {X 0,Y 242.428,Z 379.599,A -85,B 0,C 180,E1 11556.65,E2 11556.65} C_VEL
LIN {X 0,Y 238.162,Z 400.412,A -85,B 0,C 180,E1 11552.016,E2 11552.016} C_VEL
LIN {X 0,Y 240.745,Z 437.726,A -85,B 0,C 180,E1 11549.768,E2 11549.768} C_VEL
LIN {X 0,Y 241.248,Z 446.467,A -85,B 0,C 180,E1 11549.257,E2 11549.257} C_VEL
LIN {X 0,Y 234.916,Z 540.258,A -85,B 0,C 180,E1 11544.522,E2 11544.522} C_VEL
LIN {X 0,Y 233.615,Z 558.871,A -85,B 0,C 180,E1 11543.117,E2 11543.117} C_VEL
LIN {X 0,Y 232.155,Z 576.206,A -85,B 0,C 180,E1 11541.344,E2 11541.344} C_VEL
LIN {X 0,Y 230.566,Z 593.085,A -85,B 0,C 180,E1 11539.107,E2 11539.107} C_VEL
LIN {X 0,Y 229.061,Z 608.69,A -85,B 0,C 180,E1 11536.479,E2 11536.479} C_VEL
LIN {X 0,Y 227.751,Z 622.914,A -85,B 0,C 180,E1 11533.451,E2 11533.451} C_VEL
LIN {X 0,Y 226.815,Z 635.305,A -85,B 0,C 180,E1 11530.152,E2 11530.152} C_VEL
LIN {X 0,Y 226.343,Z 645.301,A -85,B 0,C 180,E1 11526.846,E2 11526.846} C_VEL
LIN {X 0,Y 226.321,Z 654.07,A -85,B 0,C 180,E1 11523.171,E2 11523.171} C_VEL
LIN {X 0,Y 226.901,Z 661.166,A -85,B 0,C 180,E1 11519.239,E2 11519.239} C_VEL
LIN {X 0,Y 228.125,Z 666.059,A -85,B 0,C 180,E1 11515.472,E2 11515.472} C_VEL
LIN {X 0,Y 230.278,Z 669.304,A -85,B 0,C 180,E1 11511.507,E2 11511.507} C_VEL
LIN {X 0,Y 233.154,Z 670.628,A -85,B 0,C 180,E1 11507.867,E2 11507.867} C_VEL
LIN {X 0,Y 237.176,Z 670.178,A -85,B 0,C 180,E1 11504.093,E2 11504.093} C_VEL
LIN {X 0,Y 242.207,Z 667.972,A -85,B 0,C 180,E1 11500.462,E2 11500.462} C_VEL
LIN {X 0,Y 245.696,Z 665.742,A -85,B 0,C 180,E1 11498.357,E2 11498.357} C_VEL
LIN {X 0,Y 247.943,Z 663.855,A -85,B 0,C 180,E1 11496.547,E2 11496.547} C_VEL
LIN {X 0,Y 251.171,Z 659.887,A -85,B 0,C 180,E1 11492.485,E2 11492.485} C_VEL
LIN {X 0,Y 253.843,Z 657.294,A -85,B 0,C 180,E1 11490.954,E2 11490.954} C_VEL
LIN {X 0,Y 254.356,Z 656.845,A -85,B 0,C 180,E1 11490.758,E2 11490.758} C_VEL
LIN {X 0,Y 263.686,Z 647.947,A -85,B 0,C 180,E1 11487.677,E2 11487.677} C_VEL
LIN {X 0,Y 273.142,Z 637.793,A -85,B 0,C 180,E1 11485.084,E2 11485.084} C_VEL
LIN {X 0,Y 283.629,Z 625.05,A -85,B 0,C 180,E1 11482.672,E2 11482.672} C_VEL
LIN {X 0,Y 293.304,Z 611.642,A -85,B 0,C 180,E1 11480.773,E2 11480.773} C_VEL
LIN {X 0,Y 294.229,Z 610.268,A -85,B 0,C 180,E1 11480.587,E2 11480.587} C_VEL
LIN {X 0,Y 283.845,Z 627.156,A -85,B 0,C 180,E1 11479.079,E2 11479.079} C_VEL
LIN {X 0,Y 273.665,Z 642.123,A -85,B 0,C 180,E1 11477.256,E2 11477.256} C_VEL
LIN {X 0,Y 262.583,Z 657.159,A -85,B 0,C 180,E1 11474.786,E2 11474.786} C_VEL
LIN {X 0,Y 251.999,Z 670.804,A -85,B 0,C 180,E1 11471.805,E2 11471.805} C_VEL
LIN {X 0,Y 242.187,Z 683.123,A -85,B 0,C 180,E1 11468.265,E2 11468.265} C_VEL
LIN {X 0,Y 233.466,Z 694.024,A -85,B 0,C 180,E1 11464.129,E2 11464.129} C_VEL
LIN {X 0,Y 226.251,Z 703.488,A -85,B 0,C 180,E1 11459.378,E2 11459.378} C_VEL
LIN {X 0,Y 221.113,Z 711.074,A -85,B 0,C 180,E1 11454.301,E2 11454.301} C_VEL
LIN {X 0,Y 218.056,Z 716.84,A -85,B 0,C 180,E1 11449.001,E2 11449.001} C_VEL
LIN {X 0,Y 217.006,Z 720.831,A -85,B 0,C 180,E1 11443.535,E2 11443.535} C_VEL
LIN {X 0,Y 217.649,Z 722.848,A -85,B 0,C 180,E1 11438.189,E2 11438.189} C_VEL
LIN {X 0,Y 219.012,Z 722.912,A -85,B 0,C 180,E1 11433.666,E2 11433.666} C_VEL
LIN {X 0,Y 219.887,Z 721.699,A -85,B 0,C 180,E1 11430.263,E2 11430.263} C_VEL
LIN {X 0,Y 219.816,Z 719.412,A -85,B 0,C 180,E1 11427.134,E2 11427.134} C_VEL
LIN {X 0,Y 219.169,Z 715.162,A -85,B 0,C 180,E1 11423.453,E2 11423.453} C_VEL
LIN {X 0,Y 218.569,Z 708.829,A -85,B 0,C 180,E1 11419.459,E2 11419.459} C_VEL
LIN {X 0,Y 218.494,Z 700.528,A -85,B 0,C 180,E1 11415.425,E2 11415.425} C_VEL
LIN {X 0,Y 219.087,Z 690.772,A -85,B 0,C 180,E1 11411.648,E2 11411.648} C_VEL
LIN {X 0,Y 220.426,Z 678.667,A -85,B 0,C 180,E1 11407.886,E2 11407.886} C_VEL
LIN {X 0,Y 222.383,Z 664.914,A -85,B 0,C 180,E1 11404.431,E2 11404.431} C_VEL
LIN {X 0,Y 224.717,Z 650.156,A -85,B 0,C 180,E1 11401.433,E2 11401.433} C_VEL
LIN {X 0,Y 227.228,Z 634.362,A -85,B 0,C 180,E1 11398.869,E2 11398.869} C_VEL
LIN {X 0,Y 229.829,Z 617.016,A -85,B 0,C 180,E1 11396.65,E2 11396.65} C_VEL
LIN {X 0,Y 232.205,Z 599.28,A -85,B 0,C 180,E1 11394.902,E2 11394.902} C_VEL
LIN {X 0,Y 234.167,Z 580.749,A -85,B 0,C 180,E1 11393.566,E2 11393.566} C_VEL
LIN {X 0,Y 235.697,Z 557.115,A -85,B 0,C 180,E1 11392.427,E2 11392.427} C_VEL
LIN {X 0,Y 244.162,Z 426.898,A -85,B 0,C 180,E1 11387.036,E2 11387.036} C_VEL
LIN {X 0,Y 242.695,Z 395.213,A -85,B 0,C 180,E1 11385.398,E2 11385.398} C_VEL
LIN {X 0,Y 241.077,Z 391.201,A -85,B 0,C 180,E1 11385.007,E2 11385.007} C_VEL
LIN {X 0,Y 234.98,Z 371.357,A -85,B 0,C 180,E1 11379.983,E2 11379.983} C_VEL
LIN {X 0,Y 229.455,Z 354.187,A -85,B 0,C 180,E1 11375.117,E2 11375.117} C_VEL
LIN {X 0,Y 224.256,Z 338.786,A -85,B 0,C 180,E1 11370.256,E2 11370.256} C_VEL
LIN {X 0,Y 219.794,Z 326.408,A -85,B 0,C 180,E1 11365.898,E2 11365.898} C_VEL
LIN {X 0,Y 218.85,Z 323.54,A -85,B 0,C 180,E1 11364.786,E2 11364.786} C_VEL
LIN {X 0,Y 218.867,Z 323.536,A -85,B 0,C 180,E1 11359.484,E2 11359.484} C_VEL
LIN {X 0,Y 218.86,Z 323.532,A -85,B 0,C 180,E1 11354.016,E2 11354.016} C_VEL
LIN {X 0,Y 218.848,Z 323.528,A -85,B 0,C 180,E1 11348.675,E2 11348.675} C_VEL
LIN {X 0,Y 218.862,Z 323.527,A -85,B 0,C 180,E1 11343.408,E2 11343.408} C_VEL
LIN {X 0,Y 218.863,Z 323.526,A -85,B 0,C 180,E1 11337.909,E2 11337.909} C_VEL
LIN {X 0,Y 218.855,Z 323.534,A -85,B 0,C 180,E1 11332.655,E2 11332.655} C_VEL
LIN {X 0,Y 218.873,Z 323.531,A -85,B 0,C 180,E1 11327.338,E2 11327.338} C_VEL
LIN {X 0,Y 218.868,Z 323.519,A -85,B 0,C 180,E1 11321.836,E2 11321.836} C_VEL
LIN {X 0,Y 218.861,Z 323.534,A -85,B 0,C 180,E1 11316.585,E2 11316.585} C_VEL
LIN {X 0,Y 218.881,Z 323.509,A -85,B 0,C 180,E1 11311.286,E2 11311.286} C_VEL
LIN {X 0,Y 218.874,Z 323.532,A -85,B 0,C 180,E1 11305.772,E2 11305.772} C_VEL
LIN {X 0,Y 218.862,Z 323.517,A -85,B 0,C 180,E1 11300.536,E2 11300.536} C_VEL
LIN {X 0,Y 218.878,Z 323.527,A -85,B 0,C 180,E1 11295.299,E2 11295.299} C_VEL
LIN {X 0,Y 218.877,Z 323.522,A -85,B 0,C 180,E1 11289.755,E2 11289.755} C_VEL
LIN {X 0,Y 218.869,Z 323.521,A -85,B 0,C 180,E1 11284.502,E2 11284.502} C_VEL
LIN {X 0,Y 218.896,Z 323.529,A -85,B 0,C 180,E1 11279.256,E2 11279.256} C_VEL
LIN {X 0,Y 218.879,Z 323.508,A -85,B 0,C 180,E1 11273.7,E2 11273.7} C_VEL
LIN {X 0,Y 218.877,Z 323.532,A -85,B 0,C 180,E1 11268.647,E2 11268.647} C_VEL
LIN {X 0,Y 218.889,Z 323.512,A -85,B 0,C 180,E1 11263.2,E2 11263.2} C_VEL
LIN {X 0,Y 218.884,Z 323.534,A -85,B 0,C 180,E1 11257.61,E2 11257.61} C_VEL
LIN {X 0,Y 218.873,Z 323.526,A -85,B 0,C 180,E1 11252.354,E2 11252.354} C_VEL
LIN {X 0,Y 218.886,Z 323.522,A -85,B 0,C 180,E1 11247.118,E2 11247.118} C_VEL
LIN {X 0,Y 218.886,Z 323.532,A -85,B 0,C 180,E1 11241.593,E2 11241.593} C_VEL
LIN {X 0,Y 218.876,Z 323.533,A -85,B 0,C 180,E1 11236.256,E2 11236.256} C_VEL
LIN {X 0,Y 218.897,Z 323.531,A -85,B 0,C 180,E1 11230.985,E2 11230.985} C_VEL
LIN {X 0,Y 218.89,Z 323.529,A -85,B 0,C 180,E1 11225.436,E2 11225.436} C_VEL
LIN {X 0,Y 218.884,Z 323.534,A -85,B 0,C 180,E1 11220.136,E2 11220.136} C_VEL
LIN {X 0,Y 218.893,Z 323.599,A -85,B 0,C 180,E1 11216.228,E2 11216.228} C_VEL
LIN {X 0,Y 223.13,Z 336.973,A -85,B 0,C 180,E1 11211.143,E2 11211.143} C_VEL
LIN {X 0,Y 227.077,Z 350.554,A -85,B 0,C 180,E1 11206.439,E2 11206.439} C_VEL
LIN {X 0,Y 230.914,Z 365.093,A -85,B 0,C 180,E1 11201.816,E2 11201.816} C_VEL
LIN {X 0,Y 234.64,Z 380.936,A -85,B 0,C 180,E1 11197.167,E2 11197.167} C_VEL
LIN {X 0,Y 230.642,Z 400.212,A -85,B 0,C 180,E1 11192.729,E2 11192.729} C_VEL
LIN {X 0,Y 232.911,Z 436.013,A -85,B 0,C 180,E1 11190.493,E2 11190.493} C_VEL
LIN {X 0,Y 233.597,Z 446.917,A -85,B 0,C 180,E1 11189.826,E2 11189.826} C_VEL
LIN {X 0,Y 227.062,Z 540.782,A -85,B 0,C 180,E1 11184.906,E2 11184.906} C_VEL
LIN {X 0,Y 225.751,Z 559.058,A -85,B 0,C 180,E1 11183.487,E2 11183.487} C_VEL
LIN {X 0,Y 224.291,Z 576.009,A -85,B 0,C 180,E1 11181.711,E2 11181.711} C_VEL
LIN {X 0,Y 222.573,Z 593.758,A -85,B 0,C 180,E1 11179.275,E2 11179.275} C_VEL
LIN {X 0,Y 221.035,Z 609.355,A -85,B 0,C 180,E1 11176.554,E2 11176.554} C_VEL
LIN {X 0,Y 219.663,Z 624.244,A -85,B 0,C 180,E1 11173.285,E2 11173.285} C_VEL
LIN {X 0,Y 218.773,Z 636.2,A -85,B 0,C 180,E1 11169.997,E2 11169.997} C_VEL
LIN {X 0,Y 218.322,Z 646.208,A -85,B 0,C 180,E1 11166.57,E2 11166.57} C_VEL
LIN {X 0,Y 218.345,Z 654.846,A -85,B 0,C 180,E1 11162.883,E2 11162.883} C_VEL
LIN {X 0,Y 218.906,Z 661.505,A -85,B 0,C 180,E1 11159.211,E2 11159.211} C_VEL
LIN {X 0,Y 220.296,Z 667.063,A -85,B 0,C 180,E1 11155.049,E2 11155.049} C_VEL
LIN {X 0,Y 222.445,Z 670.41,A -85,B 0,C 180,E1 11151.206,E2 11151.206} C_VEL
LIN {X 0,Y 225.709,Z 672.158,A -85,B 0,C 180,E1 11147.2,E2 11147.2} C_VEL
LIN {X 0,Y 230.028,Z 672.096,A -85,B 0,C 180,E1 11143.325,E2 11143.325} C_VEL
LIN {X 0,Y 235.749,Z 670.04,A -85,B 0,C 180,E1 11139.386,E2 11139.386} C_VEL
LIN {X 0,Y 242.198,Z 666.346,A -85,B 0,C 180,E1 11135.874,E2 11135.874} C_VEL
LIN {X 0,Y 250.112,Z 660.429,A -85,B 0,C 180,E1 11132.369,E2 11132.369} C_VEL
LIN {X 0,Y 254.356,Z 656.845,A -85,B 0,C 180,E1 11130.758,E2 11130.758} C_VEL
LIN {X 0,Y 257.538,Z 653.937,A -85,B 0,C 180,E1 11129.308,E2 11129.308} C_VEL
LIN {X 0,Y 263.697,Z 647.52,A -85,B 0,C 180,E1 11125.627,E2 11125.627} C_VEL
LIN {X 0,Y 267.173,Z 643.907,A -85,B 0,C 180,E1 11124.367,E2 11124.367} C_VEL
LIN {X 0,Y 267.762,Z 643.304,A -85,B 0,C 180,E1 11124.216,E2 11124.216} C_VEL
LIN {X 0,Y 278.457,Z 631.864,A -85,B 0,C 180,E1 11121.856,E2 11121.856} C_VEL
LIN {X 0,Y 283.42,Z 626.062,A -85,B 0,C 180,E1 11120.873,E2 11120.873} C_VEL
LIN {X 0,Y 272.401,Z 641.046,A -85,B 0,C 180,E1 11119.126,E2 11119.126} C_VEL
LIN {X 0,Y 260.661,Z 655.742,A -85,B 0,C 180,E1 11116.789,E2 11116.789} C_VEL
LIN {X 0,Y 249.342,Z 669.093,A -85,B 0,C 180,E1 11113.928,E2 11113.928} C_VEL
LIN {X 0,Y 238.703,Z 681.168,A -85,B 0,C 180,E1 11110.487,E2 11110.487} C_VEL
LIN {X 0,Y 229.078,Z 691.898,A -85,B 0,C 180,E1 11106.415,E2 11106.415} C_VEL
LIN {X 0,Y 220.895,Z 701.272,A -85,B 0,C 180,E1 11101.675,E2 11101.675} C_VEL
LIN {X 0,Y 214.595,Z 709.177,A -85,B 0,C 180,E1 11096.274,E2 11096.274} C_VEL
LIN {X 0,Y 210.811,Z 714.911,A -85,B 0,C 180,E1 11090.84,E2 11090.84} C_VEL
LIN {X 0,Y 209.154,Z 719.063,A -85,B 0,C 180,E1 11084.962,E2 11084.962} C_VEL
LIN {X 0,Y 209.509,Z 721.106,A -85,B 0,C 180,E1 11079.34,E2 11079.34} C_VEL
LIN {X 0,Y 210.869,Z 721.274,A -85,B 0,C 180,E1 11074.626,E2 11074.626} C_VEL
LIN {X 0,Y 212.006,Z 720.096,A -85,B 0,C 180,E1 11070.907,E2 11070.907} C_VEL
LIN {X 0,Y 212.125,Z 718.058,A -85,B 0,C 180,E1 11067.878,E2 11067.878} C_VEL
LIN {X 0,Y 211.532,Z 714.202,A -85,B 0,C 180,E1 11064.305,E2 11064.305} C_VEL
LIN {X 0,Y 210.835,Z 708.046,A -85,B 0,C 180,E1 11060.172,E2 11060.172} C_VEL
LIN {X 0,Y 210.643,Z 699.908,A -85,B 0,C 180,E1 11055.993,E2 11055.993} C_VEL
LIN {X 0,Y 211.135,Z 690.313,A -85,B 0,C 180,E1 11052.075,E2 11052.075} C_VEL
LIN {X 0,Y 212.277,Z 679.383,A -85,B 0,C 180,E1 11048.447,E2 11048.447} C_VEL
LIN {X 0,Y 214.128,Z 665.993,A -85,B 0,C 180,E1 11044.857,E2 11044.857} C_VEL
LIN {X 0,Y 216.575,Z 650.569,A -85,B 0,C 180,E1 11041.528,E2 11041.528} C_VEL
LIN {X 0,Y 219.126,Z 634.832,A -85,B 0,C 180,E1 11038.811,E2 11038.811} C_VEL
LIN {X 0,Y 221.759,Z 617.684,A -85,B 0,C 180,E1 11036.492,E2 11036.492} C_VEL
LIN {X 0,Y 224.281,Z 599.359,A -85,B 0,C 180,E1 11034.584,E2 11034.584} C_VEL
LIN {X 0,Y 226.316,Z 580.89,A -85,B 0,C 180,E1 11033.171,E2 11033.171} C_VEL
LIN {X 0,Y 227.857,Z 558.227,A -85,B 0,C 180,E1 11032.009,E2 11032.009} C_VEL
LIN {X 0,Y 236.683,Z 427.335,A -85,B 0,C 180,E1 11026.35,E2 11026.35} C_VEL
LIN {X 0,Y 235.336,Z 397.508,A -85,B 0,C 180,E1 11024.748,E2 11024.748} C_VEL
LIN {X 0,Y 232.76,Z 391.202,A -85,B 0,C 180,E1 11024.102,E2 11024.102} C_VEL
LIN {X 0,Y 227.217,Z 373.011,A -85,B 0,C 180,E1 11019.325,E2 11019.325} C_VEL
LIN {X 0,Y 221.921,Z 356.436,A -85,B 0,C 180,E1 11014.466,E2 11014.466} C_VEL
LIN {X 0,Y 217.161,Z 342.231,A -85,B 0,C 180,E1 11009.822,E2 11009.822} C_VEL
LIN {X 0,Y 212.707,Z 329.863,A -85,B 0,C 180,E1 11005.329,E2 11005.329} C_VEL
LIN {X 0,Y 210.917,Z 324.525,A -85,B 0,C 180,E1 11003.174,E2 11003.174} C_VEL
LIN {X 0,Y 210.926,Z 324.52,A -85,B 0,C 180,E1 10997.664,E2 10997.664} C_VEL
LIN {X 0,Y 210.917,Z 324.521,A -85,B 0,C 180,E1 10992.043,E2 10992.043} C_VEL
LIN {X 0,Y 210.913,Z 324.526,A -85,B 0,C 180,E1 10986.81,E2 10986.81} C_VEL
LIN {X 0,Y 210.929,Z 324.523,A -85,B 0,C 180,E1 10981.362,E2 10981.362} C_VEL
LIN {X 0,Y 210.926,Z 324.516,A -85,B 0,C 180,E1 10975.654,E2 10975.654} C_VEL
LIN {X 0,Y 210.917,Z 324.51,A -85,B 0,C 180,E1 10970.178,E2 10970.178} C_VEL
LIN {X 0,Y 210.924,Z 324.524,A -85,B 0,C 180,E1 10964.892,E2 10964.892} C_VEL
LIN {X 0,Y 210.937,Z 324.507,A -85,B 0,C 180,E1 10959.47,E2 10959.47} C_VEL
LIN {X 0,Y 210.925,Z 324.522,A -85,B 0,C 180,E1 10954.149,E2 10954.149} C_VEL
LIN {X 0,Y 210.93,Z 324.507,A -85,B 0,C 180,E1 10948.895,E2 10948.895} C_VEL
LIN {X 0,Y 210.939,Z 324.518,A -85,B 0,C 180,E1 10943.333,E2 10943.333} C_VEL
LIN {X 0,Y 210.938,Z 324.498,A -85,B 0,C 180,E1 10937.681,E2 10937.681} C_VEL
LIN {X 0,Y 210.928,Z 324.521,A -85,B 0,C 180,E1 10932.305,E2 10932.305} C_VEL
LIN {X 0,Y 210.936,Z 324.491,A -85,B 0,C 180,E1 10927.01,E2 10927.01} C_VEL
LIN {X 0,Y 210.95,Z 324.521,A -85,B 0,C 180,E1 10921.422,E2 10921.422} C_VEL
LIN {X 0,Y 210.936,Z 324.499,A -85,B 0,C 180,E1 10915.852,E2 10915.852} C_VEL
LIN {X 0,Y 210.935,Z 324.519,A -85,B 0,C 180,E1 10910.532,E2 10910.532} C_VEL
LIN {X 0,Y 210.953,Z 324.504,A -85,B 0,C 180,E1 10905.108,E2 10905.108} C_VEL
LIN {X 0,Y 210.944,Z 324.521,A -85,B 0,C 180,E1 10899.547,E2 10899.547} C_VEL
LIN {X 0,Y 210.93,Z 324.505,A -85,B 0,C 180,E1 10894.348,E2 10894.348} C_VEL
LIN {X 0,Y 210.95,Z 324.519,A -85,B 0,C 180,E1 10888.912,E2 10888.912} C_VEL
LIN {X 0,Y 210.964,Z 324.519,A -85,B 0,C 180,E1 10883.193,E2 10883.193} C_VEL
LIN {X 0,Y 210.948,Z 324.518,A -85,B 0,C 180,E1 10877.505,E2 10877.505} C_VEL
LIN {X 0,Y 210.943,Z 324.519,A -85,B 0,C 180,E1 10872.296,E2 10872.296} C_VEL
LIN {X 0,Y 210.96,Z 324.522,A -85,B 0,C 180,E1 10866.833,E2 10866.833} C_VEL
LIN {X 0,Y 210.968,Z 324.516,A -85,B 0,C 180,E1 10861.089,E2 10861.089} C_VEL
LIN {X 0,Y 210.971,Z 324.675,A -85,B 0,C 180,E1 10857.617,E2 10857.617} C_VEL
LIN {X 0,Y 215.236,Z 337.902,A -85,B 0,C 180,E1 10852.345,E2 10852.345} C_VEL
LIN {X 0,Y 219.255,Z 351.686,A -85,B 0,C 180,E1 10847.373,E2 10847.373} C_VEL
LIN {X 0,Y 223.243,Z 366.931,A -85,B 0,C 180,E1 10842.351,E2 10842.351} C_VEL
LIN {X 0,Y 226.951,Z 382.871,A -85,B 0,C 180,E1 10837.53,E2 10837.53} C_VEL
LIN {X 0,Y 223.151,Z 400.199,A -85,B 0,C 180,E1 10833.469,E2 10833.469} C_VEL
LIN {X 0,Y 225.219,Z 435.678,A -85,B 0,C 180,E1 10831.174,E2 10831.174} C_VEL
LIN {X 0,Y 225.949,Z 447.522,A -85,B 0,C 180,E1 10830.42,E2 10830.42} C_VEL
LIN {X 0,Y 219.253,Z 540.462,A -85,B 0,C 180,E1 10825.347,E2 10825.347} C_VEL
LIN {X 0,Y 217.846,Z 559.451,A -85,B 0,C 180,E1 10823.817,E2 10823.817} C_VEL
LIN {X 0,Y 216.241,Z 577.431,A -85,B 0,C 180,E1 10821.848,E2 10821.848} C_VEL
LIN {X 0,Y 214.584,Z 594.294,A -85,B 0,C 180,E1 10819.456,E2 10819.456} C_VEL
LIN {X 0,Y 212.944,Z 610.673,A -85,B 0,C 180,E1 10816.499,E2 10816.499} C_VEL
LIN {X 0,Y 211.622,Z 624.859,A -85,B 0,C 180,E1 10813.263,E2 10813.263} C_VEL
LIN {X 0,Y 210.681,Z 637.797,A -85,B 0,C 180,E1 10809.557,E2 10809.557} C_VEL
LIN {X 0,Y 210.293,Z 647.778,A -85,B 0,C 180,E1 10806,E2 10806} C_VEL
LIN {X 0,Y 210.409,Z 656.375,A -85,B 0,C 180,E1 10802.175,E2 10802.175} C_VEL
LIN {X 0,Y 211.18,Z 663.399,A -85,B 0,C 180,E1 10798.097,E2 10798.097} C_VEL
LIN {X 0,Y 212.731,Z 668.579,A -85,B 0,C 180,E1 10794.061,E2 10794.061} C_VEL
LIN {X 0,Y 215.365,Z 672.135,A -85,B 0,C 180,E1 10789.835,E2 10789.835} C_VEL
LIN {X 0,Y 219.077,Z 673.87,A -85,B 0,C 180,E1 10785.729,E2 10785.729} C_VEL
LIN {X 0,Y 223.897,Z 673.802,A -85,B 0,C 180,E1 10781.781,E2 10781.781} C_VEL
LIN {X 0,Y 230.201,Z 671.825,A -85,B 0,C 180,E1 10777.794,E2 10777.794} C_VEL
LIN {X 0,Y 237.225,Z 668.257,A -85,B 0,C 180,E1 10774.267,E2 10774.267} C_VEL
LIN {X 0,Y 245.768,Z 662.531,A -85,B 0,C 180,E1 10770.775,E2 10770.775} C_VEL
LIN {X 0,Y 254.809,Z 655.379,A -85,B 0,C 180,E1 10767.744,E2 10767.744} C_VEL
LIN {X 0,Y 265.395,Z 645.645,A -85,B 0,C 180,E1 10764.798,E2 10764.798} C_VEL
LIN {X 0,Y 267.762,Z 643.304,A -85,B 0,C 180,E1 10764.216,E2 10764.216} C_VEL
LIN {X 0,Y 268.745,Z 642.365,A -85,B 0,C 180,E1 10763.726,E2 10763.726} C_VEL
LIN {X 0,Y 268.9,Z 642.438,A -85,B 0,C 180,E1 10762.927,E2 10762.927} C_VEL
LIN {X 0,Y 267.839,Z 643.966,A -85,B 0,C 180,E1 10761.884,E2 10761.884} C_VEL
LIN {X 0,Y 265.476,Z 646.963,A -85,B 0,C 180,E1 10760.804,E2 10760.804} C_VEL
LIN {X 0,Y 260.372,Z 653.166,A -85,B 0,C 180,E1 10759.201,E2 10759.201} C_VEL
LIN {X 0,Y 255.609,Z 658.565,A -85,B 0,C 180,E1 10758.058,E2 10758.058} C_VEL
LIN {X 0,Y 243.155,Z 671.771,A -85,B 0,C 180,E1 10755.015,E2 10755.015} C_VEL
LIN {X 0,Y 231.602,Z 683.53,A -85,B 0,C 180,E1 10751.342,E2 10751.342} C_VEL
LIN {X 0,Y 221.235,Z 693.867,A -85,B 0,C 180,E1 10746.95,E2 10746.95} C_VEL
LIN {X 0,Y 212.904,Z 702.386,A -85,B 0,C 180,E1 10742.054,E2 10742.054} C_VEL
LIN {X 0,Y 206.425,Z 709.614,A -85,B 0,C 180,E1 10736.346,E2 10736.346} C_VEL
LIN {X 0,Y 202.618,Z 714.781,A -85,B 0,C 180,E1 10730.512,E2 10730.512} C_VEL
LIN {X 0,Y 201.19,Z 718.21,A -85,B 0,C 180,E1 10724.39,E2 10724.39} C_VEL
LIN {X 0,Y 201.833,Z 719.617,A -85,B 0,C 180,E1 10718.549,E2 10718.549} C_VEL
LIN {X 0,Y 203.406,Z 719.174,A -85,B 0,C 180,E1 10713.666,E2 10713.666} C_VEL
LIN {X 0,Y 204.379,Z 717.763,A -85,B 0,C 180,E1 10710.282,E2 10710.282} C_VEL
LIN {X 0,Y 204.286,Z 715.298,A -85,B 0,C 180,E1 10707.197,E2 10707.197} C_VEL
LIN {X 0,Y 203.538,Z 710.623,A -85,B 0,C 180,E1 10703.231,E2 10703.231} C_VEL
LIN {X 0,Y 202.918,Z 703.722,A -85,B 0,C 180,E1 10698.923,E2 10698.923} C_VEL
LIN {X 0,Y 202.921,Z 694.734,A -85,B 0,C 180,E1 10694.571,E2 10694.571} C_VEL
LIN {X 0,Y 203.71,Z 684.098,A -85,B 0,C 180,E1 10690.464,E2 10690.464} C_VEL
LIN {X 0,Y 205.189,Z 671.914,A -85,B 0,C 180,E1 10686.67,E2 10686.67} C_VEL
LIN {X 0,Y 207.283,Z 658.029,A -85,B 0,C 180,E1 10683.179,E2 10683.179} C_VEL
LIN {X 0,Y 209.864,Z 642.249,A -85,B 0,C 180,E1 10679.986,E2 10679.986} C_VEL
LIN {X 0,Y 212.485,Z 626.068,A -85,B 0,C 180,E1 10677.388,E2 10677.388} C_VEL
LIN {X 0,Y 215.179,Z 608.047,A -85,B 0,C 180,E1 10675.145,E2 10675.145} C_VEL
LIN {X 0,Y 217.58,Z 589.479,A -85,B 0,C 180,E1 10673.401,E2 10673.401} C_VEL
LIN {X 0,Y 219.262,Z 570.829,A -85,B 0,C 180,E1 10672.161,E2 10672.161} C_VEL
LIN {X 0,Y 229.212,Z 427.865,A -85,B 0,C 180,E1 10665.646,E2 10665.646} C_VEL
LIN {X 0,Y 227.983,Z 399.774,A -85,B 0,C 180,E1 10664.085,E2 10664.085} C_VEL
LIN {X 0,Y 224.628,Z 391.641,A -85,B 0,C 180,E1 10663.277,E2 10663.277} C_VEL
LIN {X 0,Y 219.073,Z 373.396,A -85,B 0,C 180,E1 10658.282,E2 10658.282} C_VEL
LIN {X 0,Y 213.748,Z 356.675,A -85,B 0,C 180,E1 10653.147,E2 10653.147} C_VEL
LIN {X 0,Y 208.744,Z 341.769,A -85,B 0,C 180,E1 10648,E2 10648} C_VEL
LIN {X 0,Y 204.044,Z 328.631,A -85,B 0,C 180,E1 10642.916,E2 10642.916} C_VEL
LIN {X 0,Y 202.994,Z 325.513,A -85,B 0,C 180,E1 10641.6,E2 10641.6} C_VEL
LIN {X 0,Y 202.993,Z 325.511,A -85,B 0,C 180,E1 10635.722,E2 10635.722} C_VEL
LIN {X 0,Y 202.984,Z 325.509,A -85,B 0,C 180,E1 10629.897,E2 10629.897} C_VEL
LIN {X 0,Y 202.974,Z 325.51,A -85,B 0,C 180,E1 10624.524,E2 10624.524} C_VEL
LIN {X 0,Y 202.986,Z 325.51,A -85,B 0,C 180,E1 10619.126,E2 10619.126} C_VEL
LIN {X 0,Y 203,Z 325.512,A -85,B 0,C 180,E1 10613.5,E2 10613.5} C_VEL
LIN {X 0,Y 202.99,Z 325.505,A -85,B 0,C 180,E1 10607.776,E2 10607.776} C_VEL
LIN {X 0,Y 202.98,Z 325.502,A -85,B 0,C 180,E1 10602.518,E2 10602.518} C_VEL
LIN {X 0,Y 202.996,Z 325.511,A -85,B 0,C 180,E1 10597.077,E2 10597.077} C_VEL
LIN {X 0,Y 203.002,Z 325.485,A -85,B 0,C 180,E1 10591.466,E2 10591.466} C_VEL
LIN {X 0,Y 202.995,Z 325.51,A -85,B 0,C 180,E1 10585.838,E2 10585.838} C_VEL
LIN {X 0,Y 202.986,Z 325.491,A -85,B 0,C 180,E1 10580.555,E2 10580.555} C_VEL
LIN {X 0,Y 202.999,Z 325.505,A -85,B 0,C 180,E1 10575.172,E2 10575.172} C_VEL
LIN {X 0,Y 203.011,Z 325.493,A -85,B 0,C 180,E1 10569.362,E2 10569.362} C_VEL
LIN {X 0,Y 203.006,Z 325.5,A -85,B 0,C 180,E1 10563.476,E2 10563.476} C_VEL
LIN {X 0,Y 202.999,Z 325.503,A -85,B 0,C 180,E1 10557.896,E2 10557.896} C_VEL
LIN {X 0,Y 202.997,Z 325.495,A -85,B 0,C 180,E1 10552.591,E2 10552.591} C_VEL
LIN {X 0,Y 203.007,Z 325.506,A -85,B 0,C 180,E1 10547.176,E2 10547.176} C_VEL
LIN {X 0,Y 203.004,Z 325.499,A -85,B 0,C 180,E1 10541.36,E2 10541.36} C_VEL
LIN {X 0,Y 203.002,Z 325.499,A -85,B 0,C 180,E1 10535.651,E2 10535.651} C_VEL
LIN {X 0,Y 203,Z 325.51,A -85,B 0,C 180,E1 10529.998,E2 10529.998} C_VEL
LIN {X 0,Y 203.002,Z 325.502,A -85,B 0,C 180,E1 10524.628,E2 10524.628} C_VEL
LIN {X 0,Y 203.009,Z 325.499,A -85,B 0,C 180,E1 10519.211,E2 10519.211} C_VEL
LIN {X 0,Y 203.005,Z 325.501,A -85,B 0,C 180,E1 10513.693,E2 10513.693} C_VEL
LIN {X 0,Y 203.003,Z 325.506,A -85,B 0,C 180,E1 10508.319,E2 10508.319} C_VEL
LIN {X 0,Y 203.017,Z 325.512,A -85,B 0,C 180,E1 10502.738,E2 10502.738} C_VEL
LIN {X 0,Y 203.033,Z 325.538,A -85,B 0,C 180,E1 10499.19,E2 10499.19} C_VEL
LIN {X 0,Y 207.316,Z 338.87,A -85,B 0,C 180,E1 10493.612,E2 10493.612} C_VEL
LIN {X 0,Y 211.168,Z 351.984,A -85,B 0,C 180,E1 10488.658,E2 10488.658} C_VEL
LIN {X 0,Y 214.857,Z 365.939,A -85,B 0,C 180,E1 10483.835,E2 10483.835} C_VEL
LIN {X 0,Y 218.517,Z 381.389,A -85,B 0,C 180,E1 10478.932,E2 10478.932} C_VEL
LIN {X 0,Y 219.128,Z 384.98,A -85,B 0,C 180,E1 10477.869,E2 10477.869} C_VEL
LIN {X 0,Y 215.665,Z 400.056,A -85,B 0,C 180,E1 10474.241,E2 10474.241} C_VEL
LIN {X 0,Y 217.528,Z 435.262,A -85,B 0,C 180,E1 10471.89,E2 10471.89} C_VEL
LIN {X 0,Y 218.312,Z 448.027,A -85,B 0,C 180,E1 10471.041,E2 10471.041} C_VEL
LIN {X 0,Y 211.298,Z 542.061,A -85,B 0,C 180,E1 10465.652,E2 10465.652} C_VEL
LIN {X 0,Y 209.892,Z 560.391,A -85,B 0,C 180,E1 10464.105,E2 10464.105} C_VEL
LIN {X 0,Y 208.264,Z 578.159,A -85,B 0,C 180,E1 10462.088,E2 10462.088} C_VEL
LIN {X 0,Y 206.598,Z 594.764,A -85,B 0,C 180,E1 10459.65,E2 10459.65} C_VEL
LIN {X 0,Y 204.921,Z 611.118,A -85,B 0,C 180,E1 10456.58,E2 10456.58} C_VEL
LIN {X 0,Y 203.526,Z 626.028,A -85,B 0,C 180,E1 10453.056,E2 10453.056} C_VEL
LIN {X 0,Y 202.623,Z 638.828,A -85,B 0,C 180,E1 10449.268,E2 10449.268} C_VEL
LIN {X 0,Y 202.273,Z 649.263,A -85,B 0,C 180,E1 10445.385,E2 10445.385} C_VEL
LIN {X 0,Y 202.496,Z 657.827,A -85,B 0,C 180,E1 10441.411,E2 10441.411} C_VEL
LIN {X 0,Y 203.434,Z 664.852,A -85,B 0,C 180,E1 10437.179,E2 10437.179} C_VEL
LIN {X 0,Y 205.383,Z 670.354,A -85,B 0,C 180,E1 10432.724,E2 10432.724} C_VEL
LIN {X 0,Y 208.42,Z 673.856,A -85,B 0,C 180,E1 10428.372,E2 10428.372} C_VEL
LIN {X 0,Y 212.622,Z 675.597,A -85,B 0,C 180,E1 10424.169,E2 10424.169} C_VEL
LIN {X 0,Y 217.976,Z 675.561,A -85,B 0,C 180,E1 10420.154,E2 10420.154} C_VEL
LIN {X 0,Y 225.332,Z 673.523,A -85,B 0,C 180,E1 10415.903,E2 10415.903} C_VEL
LIN {X 0,Y 233.517,Z 669.685,A -85,B 0,C 180,E1 10412.176,E2 10412.176} C_VEL
LIN {X 0,Y 243.429,Z 663.62,A -85,B 0,C 180,E1 10408.555,E2 10408.555} C_VEL
LIN {X 0,Y 253.866,Z 655.858,A -85,B 0,C 180,E1 10405.445,E2 10405.445} C_VEL
LIN {X 0,Y 264.647,Z 646.693,A -85,B 0,C 180,E1 10402.805,E2 10402.805} C_VEL
LIN {X 0,Y 272.518,Z 639.177,A -85,B 0,C 180,E1 10401.139,E2 10401.139} C_VEL
LIN {X 0,Y 260.661,Z 652.987,A -85,B 0,C 180,E1 10399.086,E2 10399.086} C_VEL
LIN {X 0,Y 255.609,Z 658.565,A -85,B 0,C 180,E1 10398.058,E2 10398.058} C_VEL
LIN {X 0,Y 250.655,Z 663.527,A -85,B 0,C 180,E1 10397.261,E2 10397.261} C_VEL
LIN {X 0,Y 237.746,Z 674.256,A -85,B 0,C 180,E1 10395.814,E2 10395.814} C_VEL
LIN {X 0,Y 232.598,Z 678.399,A -85,B 0,C 180,E1 10394.869,E2 10394.869} C_VEL
LIN {X 0,Y 231.341,Z 679.501,A -85,B 0,C 180,E1 10394.523,E2 10394.523} C_VEL
LIN {X 0,Y 220.039,Z 689.644,A -85,B 0,C 180,E1 10390.528,E2 10390.528} C_VEL
LIN {X 0,Y 210.176,Z 698.452,A -85,B 0,C 180,E1 10385.815,E2 10385.815} C_VEL
LIN {X 0,Y 202.152,Z 705.909,A -85,B 0,C 180,E1 10380.3,E2 10380.3} C_VEL
LIN {X 0,Y 196.661,Z 711.58,A -85,B 0,C 180,E1 10374.321,E2 10374.321} C_VEL
LIN {X 0,Y 193.792,Z 715.488,A -85,B 0,C 180,E1 10368.035,E2 10368.035} C_VEL
LIN {X 0,Y 193.385,Z 717.493,A -85,B 0,C 180,E1 10361.938,E2 10361.938} C_VEL
LIN {X 0,Y 194.729,Z 717.685,A -85,B 0,C 180,E1 10356.192,E2 10356.192} C_VEL
LIN {X 0,Y 196.294,Z 716.456,A -85,B 0,C 180,E1 10351.754,E2 10351.754} C_VEL
LIN {X 0,Y 196.718,Z 714.841,A -85,B 0,C 180,E1 10349.129,E2 10349.129} C_VEL
LIN {X 0,Y 196.244,Z 711.394,A -85,B 0,C 180,E1 10345.619,E2 10345.619} C_VEL
LIN {X 0,Y 195.447,Z 705.786,A -85,B 0,C 180,E1 10341.471,E2 10341.471} C_VEL
LIN {X 0,Y 195.039,Z 697.737,A -85,B 0,C 180,E1 10336.926,E2 10336.926} C_VEL
LIN {X 0,Y 195.365,Z 688.346,A -85,B 0,C 180,E1 10332.735,E2 10332.735} C_VEL
LIN {X 0,Y 196.516,Z 676.607,A -85,B 0,C 180,E1 10328.513,E2 10328.513} C_VEL
LIN {X 0,Y 198.382,Z 663.139,A -85,B 0,C 180,E1 10324.636,E2 10324.636} C_VEL
LIN {X 0,Y 200.83,Z 648.002,A -85,B 0,C 180,E1 10321.126,E2 10321.126} C_VEL
LIN {X 0,Y 203.402,Z 632.528,A -85,B 0,C 180,E1 10318.262,E2 10318.262} C_VEL
LIN {X 0,Y 206.129,Z 615.325,A -85,B 0,C 180,E1 10315.762,E2 10315.762} C_VEL
LIN {X 0,Y 208.721,Z 597.171,A -85,B 0,C 180,E1 10313.731,E2 10313.731} C_VEL
LIN {X 0,Y 210.783,Z 578.823,A -85,B 0,C 180,E1 10312.232,E2 10312.232} C_VEL
LIN {X 0,Y 212.533,Z 553.979,A -85,B 0,C 180,E1 10310.869,E2 10310.869} C_VEL
LIN {X 0,Y 221.722,Z 428.313,A -85,B 0,C 180,E1 10304.925,E2 10304.925} C_VEL
LIN {X 0,Y 220.595,Z 401.959,A -85,B 0,C 180,E1 10303.394,E2 10303.394} C_VEL
LIN {X 0,Y 216.376,Z 391.748,A -85,B 0,C 180,E1 10302.327,E2 10302.327} C_VEL
LIN {X 0,Y 210.975,Z 373.941,A -85,B 0,C 180,E1 10297.236,E2 10297.236} C_VEL
LIN {X 0,Y 206.061,Z 358.407,A -85,B 0,C 180,E1 10292.263,E2 10292.263} C_VEL
LIN {X 0,Y 201.321,Z 344.28,A -85,B 0,C 180,E1 10287.192,E2 10287.192} C_VEL
LIN {X 0,Y 197.027,Z 332.31,A -85,B 0,C 180,E1 10282.375,E2 10282.375} C_VEL
LIN {X 0,Y 195.048,Z 326.501,A -85,B 0,C 180,E1 10279.779,E2 10279.779} C_VEL
LIN {X 0,Y 195.046,Z 326.496,A -85,B 0,C 180,E1 10273.946,E2 10273.946} C_VEL
LIN {X 0,Y 195.037,Z 326.493,A -85,B 0,C 180,E1 10268.257,E2 10268.257} C_VEL
LIN {X 0,Y 195.034,Z 326.494,A -85,B 0,C 180,E1 10262.649,E2 10262.649} C_VEL
LIN {X 0,Y 195.042,Z 326.488,A -85,B 0,C 180,E1 10257.19,E2 10257.19} C_VEL
LIN {X 0,Y 195.057,Z 326.491,A -85,B 0,C 180,E1 10251.456,E2 10251.456} C_VEL
LIN {X 0,Y 195.069,Z 326.501,A -85,B 0,C 180,E1 10245.459,E2 10245.459} C_VEL
LIN {X 0,Y 195.057,Z 326.482,A -85,B 0,C 180,E1 10239.605,E2 10239.605} C_VEL
LIN {X 0,Y 195.052,Z 326.495,A -85,B 0,C 180,E1 10233.847,E2 10233.847} C_VEL
LIN {X 0,Y 195.046,Z 326.489,A -85,B 0,C 180,E1 10228.312,E2 10228.312} C_VEL
LIN {X 0,Y 195.05,Z 326.494,A -85,B 0,C 180,E1 10222.786,E2 10222.786} C_VEL
LIN {X 0,Y 195.057,Z 326.478,A -85,B 0,C 180,E1 10217.136,E2 10217.136} C_VEL
LIN {X 0,Y 195.069,Z 326.494,A -85,B 0,C 180,E1 10211.389,E2 10211.389} C_VEL
LIN {X 0,Y 195.054,Z 326.47,A -85,B 0,C 180,E1 10205.756,E2 10205.756} C_VEL
LIN {X 0,Y 195.054,Z 326.5,A -85,B 0,C 180,E1 10200.153,E2 10200.153} C_VEL
LIN {X 0,Y 195.058,Z 326.468,A -85,B 0,C 180,E1 10194.853,E2 10194.853} C_VEL
LIN {X 0,Y 195.069,Z 326.499,A -85,B 0,C 180,E1 10189.148,E2 10189.148} C_VEL
LIN {X 0,Y 195.07,Z 326.474,A -85,B 0,C 180,E1 10183.333,E2 10183.333} C_VEL
LIN {X 0,Y 195.078,Z 326.496,A -85,B 0,C 180,E1 10177.36,E2 10177.36} C_VEL
LIN {X 0,Y 195.069,Z 326.493,A -85,B 0,C 180,E1 10171.466,E2 10171.466} C_VEL
LIN {X 0,Y 195.06,Z 326.484,A -85,B 0,C 180,E1 10165.883,E2 10165.883} C_VEL
LIN {X 0,Y 195.065,Z 326.493,A -85,B 0,C 180,E1 10160.557,E2 10160.557} C_VEL
LIN {X 0,Y 195.078,Z 326.492,A -85,B 0,C 180,E1 10154.845,E2 10154.845} C_VEL
LIN {X 0,Y 195.08,Z 326.49,A -85,B 0,C 180,E1 10148.973,E2 10148.973} C_VEL
LIN {X 0,Y 195.082,Z 326.503,A -85,B 0,C 180,E1 10143.089,E2 10143.089} C_VEL
LIN {X 0,Y 195.104,Z 326.663,A -85,B 0,C 180,E1 10140.761,E2 10140.761} C_VEL
LIN {X 0,Y 198.809,Z 338.037,A -85,B 0,C 180,E1 10135.715,E2 10135.715} C_VEL
LIN {X 0,Y 202.513,Z 350.214,A -85,B 0,C 180,E1 10130.802,E2 10130.802} C_VEL
LIN {X 0,Y 206.253,Z 364.055,A -85,B 0,C 180,E1 10125.725,E2 10125.725} C_VEL
LIN {X 0,Y 209.848,Z 378.909,A -85,B 0,C 180,E1 10120.744,E2 10120.744} C_VEL
LIN {X 0,Y 211.465,Z 386.23,A -85,B 0,C 180,E1 10118.439,E2 10118.439} C_VEL
LIN {X 0,Y 208.193,Z 399.869,A -85,B 0,C 180,E1 10115.049,E2 10115.049} C_VEL
LIN {X 0,Y 209.821,Z 434.811,A -85,B 0,C 180,E1 10112.618,E2 10112.618} C_VEL
LIN {X 0,Y 210.64,Z 448.639,A -85,B 0,C 180,E1 10111.66,E2 10111.66} C_VEL
LIN {X 0,Y 203.421,Z 542.665,A -85,B 0,C 180,E1 10106.054,E2 10106.054} C_VEL
LIN {X 0,Y 201.933,Z 561.297,A -85,B 0,C 180,E1 10104.401,E2 10104.401} C_VEL
LIN {X 0,Y 200.259,Z 578.941,A -85,B 0,C 180,E1 10102.295,E2 10102.295} C_VEL
LIN {X 0,Y 198.453,Z 596.513,A -85,B 0,C 180,E1 10099.577,E2 10099.577} C_VEL
LIN {X 0,Y 196.834,Z 612.141,A -85,B 0,C 180,E1 10096.522,E2 10096.522} C_VEL
LIN {X 0,Y 195.438,Z 627.091,A -85,B 0,C 180,E1 10092.854,E2 10092.854} C_VEL
LIN {X 0,Y 194.557,Z 639.977,A -85,B 0,C 180,E1 10088.864,E2 10088.864} C_VEL
LIN {X 0,Y 194.269,Z 649.98,A -85,B 0,C 180,E1 10085.015,E2 10085.015} C_VEL
LIN {X 0,Y 194.61,Z 659.214,A -85,B 0,C 180,E1 10080.585,E2 10080.585} C_VEL
LIN {X 0,Y 195.741,Z 666.259,A -85,B 0,C 180,E1 10076.188,E2 10076.188} C_VEL
LIN {X 0,Y 197.978,Z 671.817,A -85,B 0,C 180,E1 10071.574,E2 10071.574} C_VEL
LIN {X 0,Y 201.387,Z 675.408,A -85,B 0,C 180,E1 10067.086,E2 10067.086} C_VEL
LIN {X 0,Y 206.358,Z 677.337,A -85,B 0,C 180,E1 10062.514,E2 10062.514} C_VEL
LIN {X 0,Y 212.68,Z 677.297,A -85,B 0,C 180,E1 10058.195,E2 10058.195} C_VEL
LIN {X 0,Y 220.788,Z 675.302,A -85,B 0,C 180,E1 10053.939,E2 10053.939} C_VEL
LIN {X 0,Y 229.684,Z 671.532,A -85,B 0,C 180,E1 10050.244,E2 10050.244} C_VEL
LIN {X 0,Y 240.346,Z 665.623,A -85,B 0,C 180,E1 10046.689,E2 10046.689} C_VEL
LIN {X 0,Y 251.482,Z 658.092,A -85,B 0,C 180,E1 10043.669,E2 10043.669} C_VEL
LIN {X 0,Y 261.493,Z 650.358,A -85,B 0,C 180,E1 10041.379,E2 10041.379} C_VEL
LIN {X 0,Y 248.254,Z 663.685,A -85,B 0,C 180,E1 10038.867,E2 10038.867} C_VEL
LIN {X 0,Y 235.716,Z 675.535,A -85,B 0,C 180,E1 10035.798,E2 10035.798} C_VEL
LIN {X 0,Y 231.341,Z 679.501,A -85,B 0,C 180,E1 10034.523,E2 10034.523} C_VEL
LIN {X 0,Y 226.46,Z 683.419,A -85,B 0,C 180,E1 10033.354,E2 10033.354} C_VEL
LIN {X 0,Y 213.458,Z 691.56,A -85,B 0,C 180,E1 10030.952,E2 10030.952} C_VEL
LIN {X 0,Y 208.583,Z 694.61,A -85,B 0,C 180,E1 10029.564,E2 10029.564} C_VEL
LIN {X 0,Y 207.477,Z 695.44,A -85,B 0,C 180,E1 10029.094,E2 10029.094} C_VEL
LIN {X 0,Y 198.086,Z 702.933,A -85,B 0,C 180,E1 10023.729,E2 10023.729} C_VEL
LIN {X 0,Y 190.899,Z 709.036,A -85,B 0,C 180,E1 10017.448,E2 10017.448} C_VEL
LIN {X 0,Y 186.673,Z 713.263,A -85,B 0,C 180,E1 10010.705,E2 10010.705} C_VEL
LIN {X 0,Y 185.43,Z 715.538,A -85,B 0,C 180,E1 10003.92,E2 10003.92} C_VEL
LIN {X 0,Y 186.548,Z 715.84,A -85,B 0,C 180,E1 9997.425,E2 9997.425} C_VEL
LIN {X 0,Y 188.368,Z 714.567,A -85,B 0,C 180,E1 9992.436,E2 9992.436} C_VEL
LIN {X 0,Y 189.025,Z 713.002,A -85,B 0,C 180,E1 9989.699,E2 9989.699} C_VEL
LIN {X 0,Y 188.648,Z 709.893,A -85,B 0,C 180,E1 9986.356,E2 9986.356} C_VEL
LIN {X 0,Y 187.781,Z 704.311,A -85,B 0,C 180,E1 9982.045,E2 9982.045} C_VEL
LIN {X 0,Y 187.279,Z 696.34,A -85,B 0,C 180,E1 9977.358,E2 9977.358} C_VEL
LIN {X 0,Y 187.54,Z 686.849,A -85,B 0,C 180,E1 9972.951,E2 9972.951} C_VEL
LIN {X 0,Y 188.552,Z 675.995,A -85,B 0,C 180,E1 9968.866,E2 9968.866} C_VEL
LIN {X 0,Y 190.362,Z 662.666,A -85,B 0,C 180,E1 9964.824,E2 9964.824} C_VEL
LIN {X 0,Y 192.786,Z 647.676,A -85,B 0,C 180,E1 9961.165,E2 9961.165} C_VEL
LIN {X 0,Y 195.494,Z 631.593,A -85,B 0,C 180,E1 9958.041,E2 9958.041} C_VEL
LIN {X 0,Y 198.261,Z 614.414,A -85,B 0,C 180,E1 9955.437,E2 9955.437} C_VEL
LIN {X 0,Y 200.894,Z 596.307,A -85,B 0,C 180,E1 9953.33,E2 9953.33} C_VEL
LIN {X 0,Y 202.983,Z 577.978,A -85,B 0,C 180,E1 9951.774,E2 9951.774} C_VEL
LIN {X 0,Y 204.851,Z 552.081,A -85,B 0,C 180,E1 9950.29,E2 9950.29} C_VEL
LIN {X 0,Y 214.23,Z 428.79,A -85,B 0,C 180,E1 9944.184,E2 9944.184} C_VEL
LIN {X 0,Y 213.246,Z 404.336,A -85,B 0,C 180,E1 9942.7,E2 9942.7} C_VEL
LIN {X 0,Y 208.126,Z 391.834,A -85,B 0,C 180,E1 9941.347,E2 9941.347} C_VEL
LIN {X 0,Y 202.71,Z 373.853,A -85,B 0,C 180,E1 9935.946,E2 9935.946} C_VEL
LIN {X 0,Y 197.533,Z 357.521,A -85,B 0,C 180,E1 9930.413,E2 9930.413} C_VEL
LIN {X 0,Y 193.122,Z 344.541,A -85,B 0,C 180,E1 9925.454,E2 9925.454} C_VEL
LIN {X 0,Y 189.182,Z 333.483,A -85,B 0,C 180,E1 9920.743,E2 9920.743} C_VEL
LIN {X 0,Y 187.104,Z 327.488,A -85,B 0,C 180,E1 9917.98,E2 9917.98} C_VEL
LIN {X 0,Y 187.095,Z 327.486,A -85,B 0,C 180,E1 9912.347,E2 9912.347} C_VEL
LIN {X 0,Y 187.097,Z 327.493,A -85,B 0,C 180,E1 9906.756,E2 9906.756} C_VEL
LIN {X 0,Y 187.101,Z 327.492,A -85,B 0,C 180,E1 9900.923,E2 9900.923} C_VEL
LIN {X 0,Y 187.105,Z 327.486,A -85,B 0,C 180,E1 9895.1,E2 9895.1} C_VEL
LIN {X 0,Y 187.109,Z 327.472,A -85,B 0,C 180,E1 9889.482,E2 9889.482} C_VEL
LIN {X 0,Y 187.117,Z 327.483,A -85,B 0,C 180,E1 9883.553,E2 9883.553} C_VEL
LIN {X 0,Y 187.126,Z 327.484,A -85,B 0,C 180,E1 9877.568,E2 9877.568} C_VEL
LIN {X 0,Y 187.121,Z 327.461,A -85,B 0,C 180,E1 9871.61,E2 9871.61} C_VEL
LIN {X 0,Y 187.114,Z 327.487,A -85,B 0,C 180,E1 9865.876,E2 9865.876} C_VEL
LIN {X 0,Y 187.108,Z 327.46,A -85,B 0,C 180,E1 9860.122,E2 9860.122} C_VEL
LIN {X 0,Y 187.113,Z 327.485,A -85,B 0,C 180,E1 9854.424,E2 9854.424} C_VEL
LIN {X 0,Y 187.113,Z 327.466,A -85,B 0,C 180,E1 9848.694,E2 9848.694} C_VEL
LIN {X 0,Y 187.123,Z 327.481,A -85,B 0,C 180,E1 9842.986,E2 9842.986} C_VEL
LIN {X 0,Y 187.129,Z 327.474,A -85,B 0,C 180,E1 9837.353,E2 9837.353} C_VEL
LIN {X 0,Y 187.135,Z 327.478,A -85,B 0,C 180,E1 9831.302,E2 9831.302} C_VEL
LIN {X 0,Y 187.132,Z 327.471,A -85,B 0,C 180,E1 9825.492,E2 9825.492} C_VEL
LIN {X 0,Y 187.126,Z 327.487,A -85,B 0,C 180,E1 9819.532,E2 9819.532} C_VEL
LIN {X 0,Y 187.114,Z 327.468,A -85,B 0,C 180,E1 9813.981,E2 9813.981} C_VEL
LIN {X 0,Y 187.122,Z 327.486,A -85,B 0,C 180,E1 9808.467,E2 9808.467} C_VEL
LIN {X 0,Y 187.128,Z 327.488,A -85,B 0,C 180,E1 9802.63,E2 9802.63} C_VEL
LIN {X 0,Y 187.13,Z 327.489,A -85,B 0,C 180,E1 9796.715,E2 9796.715} C_VEL
LIN {X 0,Y 187.136,Z 327.487,A -85,B 0,C 180,E1 9790.976,E2 9790.976} C_VEL
LIN {X 0,Y 187.138,Z 327.482,A -85,B 0,C 180,E1 9785.031,E2 9785.031} C_VEL
LIN {X 0,Y 187.151,Z 327.601,A -85,B 0,C 180,E1 9782.545,E2 9782.545} C_VEL
LIN {X 0,Y 190.828,Z 338.651,A -85,B 0,C 180,E1 9777.336,E2 9777.336} C_VEL
LIN {X 0,Y 194.453,Z 350.569,A -85,B 0,C 180,E1 9772.271,E2 9772.271} C_VEL
LIN {X 0,Y 198.011,Z 363.653,A -85,B 0,C 180,E1 9767.219,E2 9767.219} C_VEL
LIN {X 0,Y 201.433,Z 377.587,A -85,B 0,C 180,E1 9762.3,E2 9762.3} C_VEL
LIN {X 0,Y 203.699,Z 387.875,A -85,B 0,C 180,E1 9758.918,E2 9758.918} C_VEL
LIN {X 0,Y 200.732,Z 399.797,A -85,B 0,C 180,E1 9755.882,E2 9755.882} C_VEL
LIN {X 0,Y 202.117,Z 433.927,A -85,B 0,C 180,E1 9753.433,E2 9753.433} C_VEL
LIN {X 0,Y 203.001,Z 449.119,A -85,B 0,C 180,E1 9752.329,E2 9752.329} C_VEL
LIN {X 0,Y 195.554,Z 542.657,A -85,B 0,C 180,E1 9746.474,E2 9746.474} C_VEL
LIN {X 0,Y 194.015,Z 561.497,A -85,B 0,C 180,E1 9744.749,E2 9744.749} C_VEL
LIN {X 0,Y 192.225,Z 579.894,A -85,B 0,C 180,E1 9742.472,E2 9742.472} C_VEL
LIN {X 0,Y 190.381,Z 597.522,A -85,B 0,C 180,E1 9739.636,E2 9739.636} C_VEL
LIN {X 0,Y 188.774,Z 612.799,A -85,B 0,C 180,E1 9736.52,E2 9736.52} C_VEL
LIN {X 0,Y 187.354,Z 627.986,A -85,B 0,C 180,E1 9732.634,E2 9732.634} C_VEL
LIN {X 0,Y 186.527,Z 640.454,A -85,B 0,C 180,E1 9728.628,E2 9728.628} C_VEL
LIN {X 0,Y 186.273,Z 650.622,A -85,B 0,C 180,E1 9724.614,E2 9724.614} C_VEL
LIN {X 0,Y 186.7,Z 659.969,A -85,B 0,C 180,E1 9719.996,E2 9719.996} C_VEL
LIN {X 0,Y 187.981,Z 667.207,A -85,B 0,C 180,E1 9715.42,E2 9715.42} C_VEL
LIN {X 0,Y 190.656,Z 673.239,A -85,B 0,C 180,E1 9710.335,E2 9710.335} C_VEL
LIN {X 0,Y 194.471,Z 676.948,A -85,B 0,C 180,E1 9705.708,E2 9705.708} C_VEL
LIN {X 0,Y 199.937,Z 679.01,A -85,B 0,C 180,E1 9701.027,E2 9701.027} C_VEL
LIN {X 0,Y 206.812,Z 679.205,A -85,B 0,C 180,E1 9696.64,E2 9696.64} C_VEL
LIN {X 0,Y 215.517,Z 677.44,A -85,B 0,C 180,E1 9692.355,E2 9692.355} C_VEL
LIN {X 0,Y 225.015,Z 674.03,A -85,B 0,C 180,E1 9688.672,E2 9688.672} C_VEL
LIN {X 0,Y 236.631,Z 668.293,A -85,B 0,C 180,E1 9685.06,E2 9685.06} C_VEL
LIN {X 0,Y 248.725,Z 660.987,A -85,B 0,C 180,E1 9682.041,E2 9682.041} C_VEL
LIN {X 0,Y 250.383,Z 659.891,A -85,B 0,C 180,E1 9681.602,E2 9681.602} C_VEL
LIN {X 0,Y 236.635,Z 671.912,A -85,B 0,C 180,E1 9678.776,E2 9678.776} C_VEL
LIN {X 0,Y 223.701,Z 682.589,A -85,B 0,C 180,E1 9675.292,E2 9675.292} C_VEL
LIN {X 0,Y 211.786,Z 692.076,A -85,B 0,C 180,E1 9671.015,E2 9671.015} C_VEL
LIN {X 0,Y 207.477,Z 695.44,A -85,B 0,C 180,E1 9669.094,E2 9669.094} C_VEL
LIN {X 0,Y 203.137,Z 698.261,A -85,B 0,C 180,E1 9667.469,E2 9667.469} C_VEL
LIN {X 0,Y 190.658,Z 703.854,A -85,B 0,C 180,E1 9663.623,E2 9663.623} C_VEL
LIN {X 0,Y 186.858,Z 705.715,A -85,B 0,C 180,E1 9661.667,E2 9661.667} C_VEL
LIN {X 0,Y 186.478,Z 705.983,A -85,B 0,C 180,E1 9661.36,E2 9661.36} C_VEL
LIN {X 0,Y 180.566,Z 710.553,A -85,B 0,C 180,E1 9654.541,E2 9654.541} C_VEL
LIN {X 0,Y 177.827,Z 713.281,A -85,B 0,C 180,E1 9647.34,E2 9647.34} C_VEL
LIN {X 0,Y 178.008,Z 714.042,A -85,B 0,C 180,E1 9640.357,E2 9640.357} C_VEL
LIN {X 0,Y 179.858,Z 713.091,A -85,B 0,C 180,E1 9634.466,E2 9634.466} C_VEL
LIN {X 0,Y 181.25,Z 711.306,A -85,B 0,C 180,E1 9630.635,E2 9630.635} C_VEL
LIN {X 0,Y 181.203,Z 708.956,A -85,B 0,C 180,E1 9627.789,E2 9627.789} C_VEL
LIN {X 0,Y 180.342,Z 704.118,A -85,B 0,C 180,E1 9623.636,E2 9623.636} C_VEL
LIN {X 0,Y 179.64,Z 697.13,A -85,B 0,C 180,E1 9619.094,E2 9619.094} C_VEL
LIN {X 0,Y 179.61,Z 687.921,A -85,B 0,C 180,E1 9614.391,E2 9614.391} C_VEL
LIN {X 0,Y 180.43,Z 677.008,A -85,B 0,C 180,E1 9609.908,E2 9609.908} C_VEL
LIN {X 0,Y 182.041,Z 664.286,A -85,B 0,C 180,E1 9605.676,E2 9605.676} C_VEL
LIN {X 0,Y 184.314,Z 649.905,A -85,B 0,C 180,E1 9601.842,E2 9601.842} C_VEL
LIN {X 0,Y 187.051,Z 633.743,A -85,B 0,C 180,E1 9598.412,E2 9598.412} C_VEL
LIN {X 0,Y 189.756,Z 617.47,A -85,B 0,C 180,E1 9595.684,E2 9595.684} C_VEL
LIN {X 0,Y 192.439,Z 599.74,A -85,B 0,C 180,E1 9593.404,E2 9593.404} C_VEL
LIN {X 0,Y 194.837,Z 580.666,A -85,B 0,C 180,E1 9591.583,E2 9591.583} C_VEL
LIN {X 0,Y 196.426,Z 561.028,A -85,B 0,C 180,E1 9590.283,E2 9590.283} C_VEL
LIN {X 0,Y 206.733,Z 429.106,A -85,B 0,C 180,E1 9583.406,E2 9583.406} C_VEL
LIN {X 0,Y 205.855,Z 406.539,A -85,B 0,C 180,E1 9581.976,E2 9581.976} C_VEL
LIN {X 0,Y 199.95,Z 392.122,A -85,B 0,C 180,E1 9580.363,E2 9580.363} C_VEL
LIN {X 0,Y 194.88,Z 375.269,A -85,B 0,C 180,E1 9575.078,E2 9575.078} C_VEL
LIN {X 0,Y 190.05,Z 359.843,A -85,B 0,C 180,E1 9569.643,E2 9569.643} C_VEL
LIN {X 0,Y 185.741,Z 346.866,A -85,B 0,C 180,E1 9564.492,E2 9564.492} C_VEL
LIN {X 0,Y 181.484,Z 334.916,A -85,B 0,C 180,E1 9559.14,E2 9559.14} C_VEL
LIN {X 0,Y 179.17,Z 328.477,A -85,B 0,C 180,E1 9555.874,E2 9555.874} C_VEL
LIN {X 0,Y 179.165,Z 328.475,A -85,B 0,C 180,E1 9549.967,E2 9549.967} C_VEL
LIN {X 0,Y 179.16,Z 328.472,A -85,B 0,C 180,E1 9544.165,E2 9544.165} C_VEL
LIN {X 0,Y 179.16,Z 328.471,A -85,B 0,C 180,E1 9538.406,E2 9538.406} C_VEL
LIN {X 0,Y 179.162,Z 328.479,A -85,B 0,C 180,E1 9532.63,E2 9532.63} C_VEL
LIN {X 0,Y 179.165,Z 328.479,A -85,B 0,C 180,E1 9526.778,E2 9526.778} C_VEL
LIN {X 0,Y 179.171,Z 328.454,A -85,B 0,C 180,E1 9521.12,E2 9521.12} C_VEL
LIN {X 0,Y 179.178,Z 328.477,A -85,B 0,C 180,E1 9515.265,E2 9515.265} C_VEL
LIN {X 0,Y 179.186,Z 328.45,A -85,B 0,C 180,E1 9509.235,E2 9509.235} C_VEL
LIN {X 0,Y 179.178,Z 328.473,A -85,B 0,C 180,E1 9503.345,E2 9503.345} C_VEL
LIN {X 0,Y 179.181,Z 328.449,A -85,B 0,C 180,E1 9497.437,E2 9497.437} C_VEL
LIN {X 0,Y 179.187,Z 328.473,A -85,B 0,C 180,E1 9491.603,E2 9491.603} C_VEL
LIN {X 0,Y 179.173,Z 328.443,A -85,B 0,C 180,E1 9485.866,E2 9485.866} C_VEL
LIN {X 0,Y 179.178,Z 328.478,A -85,B 0,C 180,E1 9480.136,E2 9480.136} C_VEL
LIN {X 0,Y 179.174,Z 328.443,A -85,B 0,C 180,E1 9474.387,E2 9474.387} C_VEL
LIN {X 0,Y 179.182,Z 328.477,A -85,B 0,C 180,E1 9468.543,E2 9468.543} C_VEL
LIN {X 0,Y 179.185,Z 328.451,A -85,B 0,C 180,E1 9462.895,E2 9462.895} C_VEL
LIN {X 0,Y 179.198,Z 328.472,A -85,B 0,C 180,E1 9457.048,E2 9457.048} C_VEL
LIN {X 0,Y 179.195,Z 328.474,A -85,B 0,C 180,E1 9450.957,E2 9450.957} C_VEL
LIN {X 0,Y 179.187,Z 328.463,A -85,B 0,C 180,E1 9444.875,E2 9444.875} C_VEL
LIN {X 0,Y 179.189,Z 328.464,A -85,B 0,C 180,E1 9439.061,E2 9439.061} C_VEL
LIN {X 0,Y 179.196,Z 328.466,A -85,B 0,C 180,E1 9433.131,E2 9433.131} C_VEL
LIN {X 0,Y 179.208,Z 328.478,A -85,B 0,C 180,E1 9426.997,E2 9426.997} C_VEL
LIN {X 0,Y 179.227,Z 328.724,A -85,B 0,C 180,E1 9424.381,E2 9424.381} C_VEL
LIN {X 0,Y 183.045,Z 339.988,A -85,B 0,C 180,E1 9418.737,E2 9418.737} C_VEL
LIN {X 0,Y 186.84,Z 352.471,A -85,B 0,C 180,E1 9413.173,E2 9413.173} C_VEL
LIN {X 0,Y 190.362,Z 365.465,A -85,B 0,C 180,E1 9407.955,E2 9407.955} C_VEL
LIN {X 0,Y 193.745,Z 379.359,A -85,B 0,C 180,E1 9402.874,E2 9402.874} C_VEL
LIN {X 0,Y 195.929,Z 389.434,A -85,B 0,C 180,E1 9399.439,E2 9399.439} C_VEL
LIN {X 0,Y 193.287,Z 399.67,A -85,B 0,C 180,E1 9396.76,E2 9396.76} C_VEL
LIN {X 0,Y 194.387,Z 432.692,A -85,B 0,C 180,E1 9394.288,E2 9394.288} C_VEL
LIN {X 0,Y 195.352,Z 449.487,A -85,B 0,C 180,E1 9393.014,E2 9393.014} C_VEL
LIN {X 0,Y 187.612,Z 543.743,A -85,B 0,C 180,E1 9386.834,E2 9386.834} C_VEL
LIN {X 0,Y 186.029,Z 562.49,A -85,B 0,C 180,E1 9385.035,E2 9385.035} C_VEL
LIN {X 0,Y 184.306,Z 579.751,A -85,B 0,C 180,E1 9382.818,E2 9382.818} C_VEL
LIN {X 0,Y 182.409,Z 597.471,A -85,B 0,C 180,E1 9379.862,E2 9379.862} C_VEL
LIN {X 0,Y 180.664,Z 613.82,A -85,B 0,C 180,E1 9376.39,E2 9376.39} C_VEL
LIN {X 0,Y 179.275,Z 628.745,A -85,B 0,C 180,E1 9372.394,E2 9372.394} C_VEL
LIN {X 0,Y 178.501,Z 640.831,A -85,B 0,C 180,E1 9368.369,E2 9368.369} C_VEL
LIN {X 0,Y 178.284,Z 651.165,A -85,B 0,C 180,E1 9364.176,E2 9364.176} C_VEL
LIN {X 0,Y 178.747,Z 660.081,A -85,B 0,C 180,E1 9359.675,E2 9359.675} C_VEL
LIN {X 0,Y 180.126,Z 667.658,A -85,B 0,C 180,E1 9354.9,E2 9354.9} C_VEL
LIN {X 0,Y 182.786,Z 673.683,A -85,B 0,C 180,E1 9349.915,E2 9349.915} C_VEL
LIN {X 0,Y 187.075,Z 678.093,A -85,B 0,C 180,E1 9344.814,E2 9344.814} C_VEL
LIN {X 0,Y 192.509,Z 680.45,A -85,B 0,C 180,E1 9340.265,E2 9340.265} C_VEL
LIN {X 0,Y 200.165,Z 681.139,A -85,B 0,C 180,E1 9335.502,E2 9335.502} C_VEL
LIN {X 0,Y 208.799,Z 680.038,A -85,B 0,C 180,E1 9331.385,E2 9331.385} C_VEL
LIN {X 0,Y 219.281,Z 676.969,A -85,B 0,C 180,E1 9327.446,E2 9327.446} C_VEL
LIN {X 0,Y 231.048,Z 672.105,A -85,B 0,C 180,E1 9323.943,E2 9323.943} C_VEL
LIN {X 0,Y 239.305,Z 667.912,A -85,B 0,C 180,E1 9321.832,E2 9321.832} C_VEL
LIN {X 0,Y 225.06,Z 678.728,A -85,B 0,C 180,E1 9318.663,E2 9318.663} C_VEL
LIN {X 0,Y 211.764,Z 688.292,A -85,B 0,C 180,E1 9314.712,E2 9314.712} C_VEL
LIN {X 0,Y 199.779,Z 696.64,A -85,B 0,C 180,E1 9309.84,E2 9309.84} C_VEL
LIN {X 0,Y 189.745,Z 703.655,A -85,B 0,C 180,E1 9303.959,E2 9303.959} C_VEL
LIN {X 0,Y 186.478,Z 705.983,A -85,B 0,C 180,E1 9301.36,E2 9301.36} C_VEL
LIN {X 0,Y 183.218,Z 707.651,A -85,B 0,C 180,E1 9299.233,E2 9299.233} C_VEL
LIN {X 0,Y 173.499,Z 710.046,A -85,B 0,C 180,E1 9294.034,E2 9294.034} C_VEL
LIN {X 0,Y 171.023,Z 710.752,A -85,B 0,C 180,E1 9291.409,E2 9291.409} C_VEL
LIN {X 0,Y 170.948,Z 710.808,A -85,B 0,C 180,E1 9291.225,E2 9291.225} C_VEL
LIN {X 0,Y 169.831,Z 712.048,A -85,B 0,C 180,E1 9283.623,E2 9283.623} C_VEL
LIN {X 0,Y 171.318,Z 711.398,A -85,B 0,C 180,E1 9276.706,E2 9276.706} C_VEL
LIN {X 0,Y 173.316,Z 709.475,A -85,B 0,C 180,E1 9271.655,E2 9271.655} C_VEL
LIN {X 0,Y 173.726,Z 707.883,A -85,B 0,C 180,E1 9269.343,E2 9269.343} C_VEL
LIN {X 0,Y 172.997,Z 703.763,A -85,B 0,C 180,E1 9265.361,E2 9265.361} C_VEL
LIN {X 0,Y 172.088,Z 697.153,A -85,B 0,C 180,E1 9260.64,E2 9260.64} C_VEL
LIN {X 0,Y 171.788,Z 688.614,A -85,B 0,C 180,E1 9255.853,E2 9255.853} C_VEL
LIN {X 0,Y 172.388,Z 677.735,A -85,B 0,C 180,E1 9250.991,E2 9250.991} C_VEL
LIN {X 0,Y 173.855,Z 665.075,A -85,B 0,C 180,E1 9246.443,E2 9246.443} C_VEL
LIN {X 0,Y 175.991,Z 651.2,A -85,B 0,C 180,E1 9242.418,E2 9242.418} C_VEL
LIN {X 0,Y 178.5,Z 636.409,A -85,B 0,C 180,E1 9238.983,E2 9238.983} C_VEL
LIN {X 0,Y 181.292,Z 619.952,A -85,B 0,C 180,E1 9235.962,E2 9235.962} C_VEL
LIN {X 0,Y 184.025,Z 602.743,A -85,B 0,C 180,E1 9233.495,E2 9233.495} C_VEL
LIN {X 0,Y 186.488,Z 584.579,A -85,B 0,C 180,E1 9231.546,E2 9231.546} C_VEL
LIN {X 0,Y 188.306,Z 564.825,A -85,B 0,C 180,E1 9230.044,E2 9230.044} C_VEL
LIN {X 0,Y 199.248,Z 429.529,A -85,B 0,C 180,E1 9222.604,E2 9222.604} C_VEL
LIN {X 0,Y 198.452,Z 408.778,A -85,B 0,C 180,E1 9221.234,E2 9221.234} C_VEL
LIN {X 0,Y 191.725,Z 392.317,A -85,B 0,C 180,E1 9219.323,E2 9219.323} C_VEL
LIN {X 0,Y 186.768,Z 375.693,A -85,B 0,C 180,E1 9213.837,E2 9213.837} C_VEL
LIN {X 0,Y 182.282,Z 361.295,A -85,B 0,C 180,E1 9208.508,E2 9208.508} C_VEL
LIN {X 0,Y 178.027,Z 348.492,A -85,B 0,C 180,E1 9203.155,E2 9203.155} C_VEL
LIN {X 0,Y 174.373,Z 338.349,A -85,B 0,C 180,E1 9198.388,E2 9198.388} C_VEL
LIN {X 0,Y 171.773,Z 331.566,A -85,B 0,C 180,E1 9194.844,E2 9194.844} C_VEL
LIN {X 0,Y 171.232,Z 329.459,A -85,B 0,C 180,E1 9193.684,E2 9193.684} C_VEL
LIN {X 0,Y 171.234,Z 329.462,A -85,B 0,C 180,E1 9187.385,E2 9187.385} C_VEL
LIN {X 0,Y 171.23,Z 329.466,A -85,B 0,C 180,E1 9181.343,E2 9181.343} C_VEL
LIN {X 0,Y 171.227,Z 329.46,A -85,B 0,C 180,E1 9175.316,E2 9175.316} C_VEL
LIN {X 0,Y 171.228,Z 329.449,A -85,B 0,C 180,E1 9169.236,E2 9169.236} C_VEL
LIN {X 0,Y 171.235,Z 329.459,A -85,B 0,C 180,E1 9163.248,E2 9163.248} C_VEL
LIN {X 0,Y 171.247,Z 329.464,A -85,B 0,C 180,E1 9157.289,E2 9157.289} C_VEL
LIN {X 0,Y 171.236,Z 329.434,A -85,B 0,C 180,E1 9151.017,E2 9151.017} C_VEL
LIN {X 0,Y 171.238,Z 329.467,A -85,B 0,C 180,E1 9145.101,E2 9145.101} C_VEL
LIN {X 0,Y 171.244,Z 329.428,A -85,B 0,C 180,E1 9139.168,E2 9139.168} C_VEL
LIN {X 0,Y 171.243,Z 329.466,A -85,B 0,C 180,E1 9133.086,E2 9133.086} C_VEL
LIN {X 0,Y 171.238,Z 329.427,A -85,B 0,C 180,E1 9126.968,E2 9126.968} C_VEL
LIN {X 0,Y 171.244,Z 329.466,A -85,B 0,C 180,E1 9120.885,E2 9120.885} C_VEL
LIN {X 0,Y 171.24,Z 329.43,A -85,B 0,C 180,E1 9114.857,E2 9114.857} C_VEL
LIN {X 0,Y 171.246,Z 329.466,A -85,B 0,C 180,E1 9108.729,E2 9108.729} C_VEL
LIN {X 0,Y 171.245,Z 329.439,A -85,B 0,C 180,E1 9102.816,E2 9102.816} C_VEL
LIN {X 0,Y 171.247,Z 329.462,A -85,B 0,C 180,E1 9096.703,E2 9096.703} C_VEL
LIN {X 0,Y 171.25,Z 329.466,A -85,B 0,C 180,E1 9090.667,E2 9090.667} C_VEL
LIN {X 0,Y 171.246,Z 329.453,A -85,B 0,C 180,E1 9084.637,E2 9084.637} C_VEL
LIN {X 0,Y 171.249,Z 329.453,A -85,B 0,C 180,E1 9078.75,E2 9078.75} C_VEL
LIN {X 0,Y 171.252,Z 329.457,A -85,B 0,C 180,E1 9072.674,E2 9072.674} C_VEL
LIN {X 0,Y 171.26,Z 329.499,A -85,B 0,C 180,E1 9066.549,E2 9066.549} C_VEL
LIN {X 0,Y 174.625,Z 339.558,A -85,B 0,C 180,E1 9061.156,E2 9061.156} C_VEL
LIN {X 0,Y 177.884,Z 349.836,A -85,B 0,C 180,E1 9056.186,E2 9056.186} C_VEL
LIN {X 0,Y 181.246,Z 361.633,A -85,B 0,C 180,E1 9051.029,E2 9051.029} C_VEL
LIN {X 0,Y 184.641,Z 375.126,A -85,B 0,C 180,E1 9045.686,E2 9045.686} C_VEL
LIN {X 0,Y 187.899,Z 389.595,A -85,B 0,C 180,E1 9040.45,E2 9040.45} C_VEL
LIN {X 0,Y 188.007,Z 391.453,A -85,B 0,C 180,E1 9039.848,E2 9039.848} C_VEL
LIN {X 0,Y 185.844,Z 399.594,A -85,B 0,C 180,E1 9037.666,E2 9037.666} C_VEL
LIN {X 0,Y 186.683,Z 431.294,A -85,B 0,C 180,E1 9035.205,E2 9035.205} C_VEL
LIN {X 0,Y 187.696,Z 449.969,A -85,B 0,C 180,E1 9033.724,E2 9033.724} C_VEL
LIN {X 0,Y 179.796,Z 543.134,A -85,B 0,C 180,E1 9027.348,E2 9027.348} C_VEL
LIN {X 0,Y 178.122,Z 562.455,A -85,B 0,C 180,E1 9025.425,E2 9025.425} C_VEL
LIN {X 0,Y 176.178,Z 581.359,A -85,B 0,C 180,E1 9022.872,E2 9022.872} C_VEL
LIN {X 0,Y 174.266,Z 598.857,A -85,B 0,C 180,E1 9019.781,E2 9019.781} C_VEL
LIN {X 0,Y 172.519,Z 615.099,A -85,B 0,C 180,E1 9016.147,E2 9016.147} C_VEL
LIN {X 0,Y 171.121,Z 630.479,A -85,B 0,C 180,E1 9011.795,E2 9011.795} C_VEL
LIN {X 0,Y 170.415,Z 642.861,A -85,B 0,C 180,E1 9007.411,E2 9007.411} C_VEL
LIN {X 0,Y 170.344,Z 653.013,A -85,B 0,C 180,E1 9003.023,E2 9003.023} C_VEL
LIN {X 0,Y 171.098,Z 662.384,A -85,B 0,C 180,E1 8997.986,E2 8997.986} C_VEL
LIN {X 0,Y 172.87,Z 669.763,A -85,B 0,C 180,E1 8993.019,E2 8993.019} C_VEL
LIN {X 0,Y 176.321,Z 675.945,A -85,B 0,C 180,E1 8987.552,E2 8987.552} C_VEL
LIN {X 0,Y 181.034,Z 679.976,A -85,B 0,C 180,E1 8982.644,E2 8982.644} C_VEL
LIN {X 0,Y 187.577,Z 682.363,A -85,B 0,C 180,E1 8977.758,E2 8977.758} C_VEL
LIN {X 0,Y 196.124,Z 683.005,A -85,B 0,C 180,E1 8973.013,E2 8973.013} C_VEL
LIN {X 0,Y 205.582,Z 681.864,A -85,B 0,C 180,E1 8968.963,E2 8968.963} C_VEL
LIN {X 0,Y 217.586,Z 678.641,A -85,B 0,C 180,E1 8964.938,E2 8964.938} C_VEL
LIN {X 0,Y 228.193,Z 674.648,A -85,B 0,C 180,E1 8962.066,E2 8962.066} C_VEL
LIN {X 0,Y 213.532,Z 684.298,A -85,B 0,C 180,E1 8958.523,E2 8958.523} C_VEL
LIN {X 0,Y 199.93,Z 692.781,A -85,B 0,C 180,E1 8954.042,E2 8954.042} C_VEL
LIN {X 0,Y 187.988,Z 699.997,A -85,B 0,C 180,E1 8948.486,E2 8948.486} C_VEL
LIN {X 0,Y 178.827,Z 705.57,A -85,B 0,C 180,E1 8942.087,E2 8942.087} C_VEL
LIN {X 0,Y 172.762,Z 709.485,A -85,B 0,C 180,E1 8934.994,E2 8934.994} C_VEL
LIN {X 0,Y 170.948,Z 710.808,A -85,B 0,C 180,E1 8931.225,E2 8931.225} C_VEL
LIN {X 0,Y 169.252,Z 711.258,A -85,B 0,C 180,E1 8928.677,E2 8928.677} C_VEL
LIN {X 0,Y 164.268,Z 710.563,A -85,B 0,C 180,E1 8923.575,E2 8923.575} C_VEL
LIN {X 0,Y 162.739,Z 709.721,A -85,B 0,C 180,E1 8920.302,E2 8920.302} C_VEL
LIN {X 0,Y 162.83,Z 709.54,A -85,B 0,C 180,E1 8919.323,E2 8919.323} C_VEL
LIN {X 0,Y 165.114,Z 707.663,A -85,B 0,C 180,E1 8913.127,E2 8913.127} C_VEL
LIN {X 0,Y 166.129,Z 705.823,A -85,B 0,C 180,E1 8910.003,E2 8910.003} C_VEL
LIN {X 0,Y 165.491,Z 702.063,A -85,B 0,C 180,E1 8906.192,E2 8906.192} C_VEL
LIN {X 0,Y 164.475,Z 695.439,A -85,B 0,C 180,E1 8901.261,E2 8901.261} C_VEL
LIN {X 0,Y 164.08,Z 686.827,A -85,B 0,C 180,E1 8896.255,E2 8896.255} C_VEL
LIN {X 0,Y 164.604,Z 676.011,A -85,B 0,C 180,E1 8891.223,E2 8891.223} C_VEL
LIN {X 0,Y 166.066,Z 663.122,A -85,B 0,C 180,E1 8886.401,E2 8886.401} C_VEL
LIN {X 0,Y 168.232,Z 649.11,A -85,B 0,C 180,E1 8882.192,E2 8882.192} C_VEL
LIN {X 0,Y 170.937,Z 633.264,A -85,B 0,C 180,E1 8878.435,E2 8878.435} C_VEL
LIN {X 0,Y 173.816,Z 616.441,A -85,B 0,C 180,E1 8875.289,E2 8875.289} C_VEL
LIN {X 0,Y 176.451,Z 599.799,A -85,B 0,C 180,E1 8872.884,E2 8872.884} C_VEL
LIN {X 0,Y 178.975,Z 580.898,A -85,B 0,C 180,E1 8870.845,E2 8870.845} C_VEL
LIN {X 0,Y 180.675,Z 561.679,A -85,B 0,C 180,E1 8869.378,E2 8869.378} C_VEL
LIN {X 0,Y 191.755,Z 429.841,A -85,B 0,C 180,E1 8861.765,E2 8861.765} C_VEL
LIN {X 0,Y 191.072,Z 411.012,A -85,B 0,C 180,E1 8860.462,E2 8860.462} C_VEL
LIN {X 0,Y 183.504,Z 392.455,A -85,B 0,C 180,E1 8858.206,E2 8858.206} C_VEL
LIN {X 0,Y 178.898,Z 376.94,A -85,B 0,C 180,E1 8852.833,E2 8852.833} C_VEL
LIN {X 0,Y 174.493,Z 362.676,A -85,B 0,C 180,E1 8847.289,E2 8847.289} C_VEL
LIN {X 0,Y 170.324,Z 350.036,A -85,B 0,C 180,E1 8841.71,E2 8841.71} C_VEL
LIN {X 0,Y 166.775,Z 340.011,A -85,B 0,C 180,E1 8836.729,E2 8836.729} C_VEL
LIN {X 0,Y 163.947,Z 332.799,A -85,B 0,C 180,E1 8832.688,E2 8832.688} C_VEL
LIN {X 0,Y 163.286,Z 330.458,A -85,B 0,C 180,E1 8831.305,E2 8831.305} C_VEL
LIN {X 0,Y 163.288,Z 330.457,A -85,B 0,C 180,E1 8825.275,E2 8825.275} C_VEL
LIN {X 0,Y 163.287,Z 330.451,A -85,B 0,C 180,E1 8818.952,E2 8818.952} C_VEL
LIN {X 0,Y 163.285,Z 330.457,A -85,B 0,C 180,E1 8812.718,E2 8812.718} C_VEL
LIN {X 0,Y 163.287,Z 330.458,A -85,B 0,C 180,E1 8806.55,E2 8806.55} C_VEL
LIN {X 0,Y 163.286,Z 330.43,A -85,B 0,C 180,E1 8800.552,E2 8800.552} C_VEL
LIN {X 0,Y 163.291,Z 330.455,A -85,B 0,C 180,E1 8794.626,E2 8794.626} C_VEL
LIN {X 0,Y 163.292,Z 330.433,A -85,B 0,C 180,E1 8788.643,E2 8788.643} C_VEL
LIN {X 0,Y 163.293,Z 330.448,A -85,B 0,C 180,E1 8782.693,E2 8782.693} C_VEL
LIN {X 0,Y 163.293,Z 330.432,A -85,B 0,C 180,E1 8776.711,E2 8776.711} C_VEL
LIN {X 0,Y 163.296,Z 330.447,A -85,B 0,C 180,E1 8770.611,E2 8770.611} C_VEL
LIN {X 0,Y 163.297,Z 330.427,A -85,B 0,C 180,E1 8764.707,E2 8764.707} C_VEL
LIN {X 0,Y 163.303,Z 330.45,A -85,B 0,C 180,E1 8758.524,E2 8758.524} C_VEL
LIN {X 0,Y 163.297,Z 330.433,A -85,B 0,C 180,E1 8752.307,E2 8752.307} C_VEL
LIN {X 0,Y 163.3,Z 330.444,A -85,B 0,C 180,E1 8746.356,E2 8746.356} C_VEL
LIN {X 0,Y 163.301,Z 330.452,A -85,B 0,C 180,E1 8740.225,E2 8740.225} C_VEL
LIN {X 0,Y 163.297,Z 330.432,A -85,B 0,C 180,E1 8734.211,E2 8734.211} C_VEL
LIN {X 0,Y 163.304,Z 330.45,A -85,B 0,C 180,E1 8728.243,E2 8728.243} C_VEL
LIN {X 0,Y 163.307,Z 330.456,A -85,B 0,C 180,E1 8722.256,E2 8722.256} C_VEL
LIN {X 0,Y 163.306,Z 330.457,A -85,B 0,C 180,E1 8716.183,E2 8716.183} C_VEL
LIN {X 0,Y 163.311,Z 330.448,A -85,B 0,C 180,E1 8709.946,E2 8709.946} C_VEL
LIN {X 0,Y 163.325,Z 330.477,A -85,B 0,C 180,E1 8708.824,E2 8708.824} C_VEL
LIN {X 0,Y 166.611,Z 340.123,A -85,B 0,C 180,E1 8703.248,E2 8703.248} C_VEL
LIN {X 0,Y 169.912,Z 350.448,A -85,B 0,C 180,E1 8697.916,E2 8697.916} C_VEL
LIN {X 0,Y 173.146,Z 361.767,A -85,B 0,C 180,E1 8692.672,E2 8692.672} C_VEL
LIN {X 0,Y 176.504,Z 374.913,A -85,B 0,C 180,E1 8687.171,E2 8687.171} C_VEL
LIN {X 0,Y 179.7,Z 389.04,A -85,B 0,C 180,E1 8681.788,E2 8681.788} C_VEL
LIN {X 0,Y 180.256,Z 392.83,A -85,B 0,C 180,E1 8680.458,E2 8680.458} C_VEL
LIN {X 0,Y 178.435,Z 399.466,A -85,B 0,C 180,E1 8678.634,E2 8678.634} C_VEL
LIN {X 0,Y 179.018,Z 429.786,A -85,B 0,C 180,E1 8676.194,E2 8676.194} C_VEL
LIN {X 0,Y 180.058,Z 450.46,A -85,B 0,C 180,E1 8674.481,E2 8674.481} C_VEL
LIN {X 0,Y 171.804,Z 544.549,A -85,B 0,C 180,E1 8667.683,E2 8667.683} C_VEL
LIN {X 0,Y 170.037,Z 564.113,A -85,B 0,C 180,E1 8665.601,E2 8665.601} C_VEL
LIN {X 0,Y 168.06,Z 582.719,A -85,B 0,C 180,E1 8662.929,E2 8662.929} C_VEL
LIN {X 0,Y 166.128,Z 600.073,A -85,B 0,C 180,E1 8659.691,E2 8659.691} C_VEL
LIN {X 0,Y 164.382,Z 616.221,A -85,B 0,C 180,E1 8655.88,E2 8655.88} C_VEL
LIN {X 0,Y 163.021,Z 631.541,A -85,B 0,C 180,E1 8651.313,E2 8651.313} C_VEL
LIN {X 0,Y 162.386,Z 643.903,A -85,B 0,C 180,E1 8646.713,E2 8646.713} C_VEL
LIN {X 0,Y 162.425,Z 654.074,A -85,B 0,C 180,E1 8642.112,E2 8642.112} C_VEL
LIN {X 0,Y 163.373,Z 663.473,A -85,B 0,C 180,E1 8636.838,E2 8636.838} C_VEL
LIN {X 0,Y 165.623,Z 671.364,A -85,B 0,C 180,E1 8631.315,E2 8631.315} C_VEL
LIN {X 0,Y 169.61,Z 677.55,A -85,B 0,C 180,E1 8625.66,E2 8625.66} C_VEL
LIN {X 0,Y 175.296,Z 681.825,A -85,B 0,C 180,E1 8620.33,E2 8620.33} C_VEL
LIN {X 0,Y 182.605,Z 684.211,A -85,B 0,C 180,E1 8615.405,E2 8615.405} C_VEL
LIN {X 0,Y 191.97,Z 684.908,A -85,B 0,C 180,E1 8610.682,E2 8610.682} C_VEL
LIN {X 0,Y 202.824,Z 683.755,A -85,B 0,C 180,E1 8606.483,E2 8606.483} C_VEL
LIN {X 0,Y 215.717,Z 680.628,A -85,B 0,C 180,E1 8602.61,E2 8602.61} C_VEL
LIN {X 0,Y 216.864,Z 680.337,A -85,B 0,C 180,E1 8602.255,E2 8602.255} C_VEL
LIN {X 0,Y 202.062,Z 688.744,A -85,B 0,C 180,E1 8598.35,E2 8598.35} C_VEL
LIN {X 0,Y 188.214,Z 696.16,A -85,B 0,C 180,E1 8593.262,E2 8593.262} C_VEL
LIN {X 0,Y 176.904,Z 702.014,A -85,B 0,C 180,E1 8587.215,E2 8587.215} C_VEL
LIN {X 0,Y 168.281,Z 706.47,A -85,B 0,C 180,E1 8579.943,E2 8579.943} C_VEL
LIN {X 0,Y 163.299,Z 709.159,A -85,B 0,C 180,E1 8571.934,E2 8571.934} C_VEL
LIN {X 0,Y 162.093,Z 709.953,A -85,B 0,C 180,E1 8563.923,E2 8563.923} C_VEL
LIN {X 0,Y 162.83,Z 709.54,A -85,B 0,C 180,E1 8559.323,E2 8559.323} C_VEL
LIN {X 0,Y 162.799,Z 708.746,A -85,B 0,C 180,E1 8556.787,E2 8556.787} C_VEL
LIN {X 0,Y 161.384,Z 706.667,A -85,B 0,C 180,E1 8553.532,E2 8553.532} C_VEL
LIN {X 0,Y 158.247,Z 701.052,A -85,B 0,C 180,E1 8547.804,E2 8547.804} C_VEL
LIN {X 0,Y 158.029,Z 700.179,A -85,B 0,C 180,E1 8547.037,E2 8547.037} C_VEL
LIN {X 0,Y 156.913,Z 693.606,A -85,B 0,C 180,E1 8541.944,E2 8541.944} C_VEL
LIN {X 0,Y 156.408,Z 684.929,A -85,B 0,C 180,E1 8536.698,E2 8536.698} C_VEL
LIN {X 0,Y 156.858,Z 674.034,A -85,B 0,C 180,E1 8531.418,E2 8531.418} C_VEL
LIN {X 0,Y 158.229,Z 661.566,A -85,B 0,C 180,E1 8526.544,E2 8526.544} C_VEL
LIN {X 0,Y 160.398,Z 647.451,A -85,B 0,C 180,E1 8522.13,E2 8522.13} C_VEL
LIN {X 0,Y 163.127,Z 631.551,A -85,B 0,C 180,E1 8518.192,E2 8518.192} C_VEL
LIN {X 0,Y 166.048,Z 614.638,A -85,B 0,C 180,E1 8514.9,E2 8514.9} C_VEL
LIN {X 0,Y 168.918,Z 596.554,A -85,B 0,C 180,E1 8512.231,E2 8512.231} C_VEL
LIN {X 0,Y 171.367,Z 577.953,A -85,B 0,C 180,E1 8510.186,E2 8510.186} C_VEL
LIN {X 0,Y 173.126,Z 557.354,A -85,B 0,C 180,E1 8508.629,E2 8508.629} C_VEL
LIN {X 0,Y 184.258,Z 430.327,A -85,B 0,C 180,E1 8500.917,E2 8500.917} C_VEL
LIN {X 0,Y 183.67,Z 413.187,A -85,B 0,C 180,E1 8499.669,E2 8499.669} C_VEL
LIN {X 0,Y 175.25,Z 392.5,A -85,B 0,C 180,E1 8496.994,E2 8496.994} C_VEL
LIN {X 0,Y 170.558,Z 376.541,A -85,B 0,C 180,E1 8491.147,E2 8491.147} C_VEL
LIN {X 0,Y 166.443,Z 363.209,A -85,B 0,C 180,E1 8485.632,E2 8485.632} C_VEL
LIN {X 0,Y 162.372,Z 350.827,A -85,B 0,C 180,E1 8479.801,E2 8479.801} C_VEL
LIN {X 0,Y 158.879,Z 341.058,A -85,B 0,C 180,E1 8474.585,E2 8474.585} C_VEL
LIN {X 0,Y 156.124,Z 334.029,A -85,B 0,C 180,E1 8470.335,E2 8470.335} C_VEL
LIN {X 0,Y 155.34,Z 331.436,A -85,B 0,C 180,E1 8468.705,E2 8468.705} C_VEL
LIN {X 0,Y 155.34,Z 331.435,A -85,B 0,C 180,E1 8462.588,E2 8462.588} C_VEL
LIN {X 0,Y 155.342,Z 331.429,A -85,B 0,C 180,E1 8456.684,E2 8456.684} C_VEL
LIN {X 0,Y 155.345,Z 331.428,A -85,B 0,C 180,E1 8450.746,E2 8450.746} C_VEL
LIN {X 0,Y 155.35,Z 331.447,A -85,B 0,C 180,E1 8444.705,E2 8444.705} C_VEL
LIN {X 0,Y 155.351,Z 331.433,A -85,B 0,C 180,E1 8438.484,E2 8438.484} C_VEL
LIN {X 0,Y 155.352,Z 331.419,A -85,B 0,C 180,E1 8432.4,E2 8432.4} C_VEL
LIN {X 0,Y 155.357,Z 331.442,A -85,B 0,C 180,E1 8426.401,E2 8426.401} C_VEL
LIN {X 0,Y 155.356,Z 331.406,A -85,B 0,C 180,E1 8419.948,E2 8419.948} C_VEL
LIN {X 0,Y 155.363,Z 331.443,A -85,B 0,C 180,E1 8413.516,E2 8413.516} C_VEL
LIN {X 0,Y 155.359,Z 331.402,A -85,B 0,C 180,E1 8407.067,E2 8407.067} C_VEL
LIN {X 0,Y 155.368,Z 331.444,A -85,B 0,C 180,E1 8400.983,E2 8400.983} C_VEL
LIN {X 0,Y 155.36,Z 331.405,A -85,B 0,C 180,E1 8394.726,E2 8394.726} C_VEL
LIN {X 0,Y 155.364,Z 331.444,A -85,B 0,C 180,E1 8388.378,E2 8388.378} C_VEL
LIN {X 0,Y 155.36,Z 331.418,A -85,B 0,C 180,E1 8382.259,E2 8382.259} C_VEL
LIN {X 0,Y 155.363,Z 331.429,A -85,B 0,C 180,E1 8375.907,E2 8375.907} C_VEL
LIN {X 0,Y 155.375,Z 331.445,A -85,B 0,C 180,E1 8369.628,E2 8369.628} C_VEL
LIN {X 0,Y 155.383,Z 331.442,A -85,B 0,C 180,E1 8362.975,E2 8362.975} C_VEL
LIN {X 0,Y 155.372,Z 331.445,A -85,B 0,C 180,E1 8356.602,E2 8356.602} C_VEL
LIN {X 0,Y 155.405,Z 331.641,A -85,B 0,C 180,E1 8351.232,E2 8351.232} C_VEL
LIN {X 0,Y 158.683,Z 340.879,A -85,B 0,C 180,E1 8345.423,E2 8345.423} C_VEL
LIN {X 0,Y 162.066,Z 351.412,A -85,B 0,C 180,E1 8339.606,E2 8339.606} C_VEL
LIN {X 0,Y 165.508,Z 363.493,A -85,B 0,C 180,E1 8333.696,E2 8333.696} C_VEL
LIN {X 0,Y 168.671,Z 376.056,A -85,B 0,C 180,E1 8328.192,E2 8328.192} C_VEL
LIN {X 0,Y 171.721,Z 389.562,A -85,B 0,C 180,E1 8322.804,E2 8322.804} C_VEL
LIN {X 0,Y 172.495,Z 394.155,A -85,B 0,C 180,E1 8321.099,E2 8321.099} C_VEL
LIN {X 0,Y 171.021,Z 399.357,A -85,B 0,C 180,E1 8319.635,E2 8319.635} C_VEL
LIN {X 0,Y 171.377,Z 428.341,A -85,B 0,C 180,E1 8317.219,E2 8317.219} C_VEL
LIN {X 0,Y 172.408,Z 450.865,A -85,B 0,C 180,E1 8315.261,E2 8315.261} C_VEL
LIN {X 0,Y 163.837,Z 545.496,A -85,B 0,C 180,E1 8308.059,E2 8308.059} C_VEL
LIN {X 0,Y 162.095,Z 564.22,A -85,B 0,C 180,E1 8305.967,E2 8305.967} C_VEL
LIN {X 0,Y 160.064,Z 582.873,A -85,B 0,C 180,E1 8303.169,E2 8303.169} C_VEL
LIN {X 0,Y 158.088,Z 600.331,A -85,B 0,C 180,E1 8299.772,E2 8299.772} C_VEL
LIN {X 0,Y 156.255,Z 617.187,A -85,B 0,C 180,E1 8295.584,E2 8295.584} C_VEL
LIN {X 0,Y 154.937,Z 632.476,A -85,B 0,C 180,E1 8290.781,E2 8290.781} C_VEL
LIN {X 0,Y 154.382,Z 644.834,A -85,B 0,C 180,E1 8285.942,E2 8285.942} C_VEL
LIN {X 0,Y 154.546,Z 655.03,A -85,B 0,C 180,E1 8281.107,E2 8281.107} C_VEL
LIN {X 0,Y 155.716,Z 664.481,A -85,B 0,C 180,E1 8275.576,E2 8275.576} C_VEL
LIN {X 0,Y 158.321,Z 672.482,A -85,B 0,C 180,E1 8269.81,E2 8269.81} C_VEL
LIN {X 0,Y 162.793,Z 678.794,A -85,B 0,C 180,E1 8263.951,E2 8263.951} C_VEL
LIN {X 0,Y 169.044,Z 683.246,A -85,B 0,C 180,E1 8258.482,E2 8258.482} C_VEL
LIN {X 0,Y 176.968,Z 685.888,A -85,B 0,C 180,E1 8253.486,E2 8253.486} C_VEL
LIN {X 0,Y 186.983,Z 686.829,A -85,B 0,C 180,E1 8248.751,E2 8248.751} C_VEL
LIN {X 0,Y 198.493,Z 686.034,A -85,B 0,C 180,E1 8244.596,E2 8244.596} C_VEL
LIN {X 0,Y 205.579,Z 684.843,A -85,B 0,C 180,E1 8242.448,E2 8242.448} C_VEL
LIN {X 0,Y 189.997,Z 692.405,A -85,B 0,C 180,E1 8237.906,E2 8237.906} C_VEL
LIN {X 0,Y 176.103,Z 698.712,A -85,B 0,C 180,E1 8232.068,E2 8232.068} C_VEL
LIN {X 0,Y 165.247,Z 703.417,A -85,B 0,C 180,E1 8225.09,E2 8225.09} C_VEL
LIN {X 0,Y 157.945,Z 706.476,A -85,B 0,C 180,E1 8217.119,E2 8217.119} C_VEL
LIN {X 0,Y 154.65,Z 707.769,A -85,B 0,C 180,E1 8208.863,E2 8208.863} C_VEL
LIN {X 0,Y 154.845,Z 707.345,A -85,B 0,C 180,E1 8200.796,E2 8200.796} C_VEL
LIN {X 0,Y 157.139,Z 705.422,A -85,B 0,C 180,E1 8194.016,E2 8194.016} C_VEL
LIN {X 0,Y 158.55,Z 703.425,A -85,B 0,C 180,E1 8190.364,E2 8190.364} C_VEL
LIN {X 0,Y 158.029,Z 700.179,A -85,B 0,C 180,E1 8187.037,E2 8187.037} C_VEL
LIN {X 0,Y 156.84,Z 697.409,A -85,B 0,C 180,E1 8184.906,E2 8184.906} C_VEL
LIN {X 0,Y 153.533,Z 692.306,A -85,B 0,C 180,E1 8181.957,E2 8181.957} C_VEL
LIN {X 0,Y 149.342,Z 684.625,A -85,B 0,C 180,E1 8178.018,E2 8178.018} C_VEL
LIN {X 0,Y 148.753,Z 681.277,A -85,B 0,C 180,E1 8176.261,E2 8176.261} C_VEL
LIN {X 0,Y 149.283,Z 670.133,A -85,B 0,C 180,E1 8170.814,E2 8170.814} C_VEL
LIN {X 0,Y 150.805,Z 657.097,A -85,B 0,C 180,E1 8165.731,E2 8165.731} C_VEL
LIN {X 0,Y 153.146,Z 642.313,A -85,B 0,C 180,E1 8161.113,E2 8161.113} C_VEL
LIN {X 0,Y 155.778,Z 627.233,A -85,B 0,C 180,E1 8157.378,E2 8157.378} C_VEL
LIN {X 0,Y 158.84,Z 609.437,A -85,B 0,C 180,E1 8153.949,E2 8153.949} C_VEL
LIN {X 0,Y 161.648,Z 591.69,A -85,B 0,C 180,E1 8151.342,E2 8151.342} C_VEL
LIN {X 0,Y 163.908,Z 573.233,A -85,B 0,C 180,E1 8149.376,E2 8149.376} C_VEL
LIN {X 0,Y 166.58,Z 540.665,A -85,B 0,C 180,E1 8147.005,E2 8147.005} C_VEL
LIN {X 0,Y 176.757,Z 430.578,A -85,B 0,C 180,E1 8140.015,E2 8140.015} C_VEL
LIN {X 0,Y 176.248,Z 415.401,A -85,B 0,C 180,E1 8138.851,E2 8138.851} C_VEL
LIN {X 0,Y 167.011,Z 392.53,A -85,B 0,C 180,E1 8135.717,E2 8135.717} C_VEL
LIN {X 0,Y 162.611,Z 377.45,A -85,B 0,C 180,E1 8129.876,E2 8129.876} C_VEL
LIN {X 0,Y 158.643,Z 364.454,A -85,B 0,C 180,E1 8124.189,E2 8124.189} C_VEL
LIN {X 0,Y 154.848,Z 352.954,A -85,B 0,C 180,E1 8118.45,E2 8118.45} C_VEL
LIN {X 0,Y 151.269,Z 342.657,A -85,B 0,C 180,E1 8112.604,E2 8112.604} C_VEL
LIN {X 0,Y 148.325,Z 335.251,A -85,B 0,C 180,E1 8107.754,E2 8107.754} C_VEL
LIN {X 0,Y 147.411,Z 332.438,A -85,B 0,C 180,E1 8105.845,E2 8105.845} C_VEL
LIN {X 0,Y 147.416,Z 332.429,A -85,B 0,C 180,E1 8099.228,E2 8099.228} C_VEL
LIN {X 0,Y 147.407,Z 332.432,A -85,B 0,C 180,E1 8092.601,E2 8092.601} C_VEL
LIN {X 0,Y 147.418,Z 332.436,A -85,B 0,C 180,E1 8085.892,E2 8085.892} C_VEL
LIN {X 0,Y 147.418,Z 332.41,A -85,B 0,C 180,E1 8079.355,E2 8079.355} C_VEL
LIN {X 0,Y 147.416,Z 332.412,A -85,B 0,C 180,E1 8072.979,E2 8072.979} C_VEL
LIN {X 0,Y 147.417,Z 332.43,A -85,B 0,C 180,E1 8066.532,E2 8066.532} C_VEL
LIN {X 0,Y 147.416,Z 332.394,A -85,B 0,C 180,E1 8060.03,E2 8060.03} C_VEL
LIN {X 0,Y 147.424,Z 332.432,A -85,B 0,C 180,E1 8053.483,E2 8053.483} C_VEL
LIN {X 0,Y 147.418,Z 332.389,A -85,B 0,C 180,E1 8046.849,E2 8046.849} C_VEL
LIN {X 0,Y 147.423,Z 332.434,A -85,B 0,C 180,E1 8040.545,E2 8040.545} C_VEL
LIN {X 0,Y 147.418,Z 332.393,A -85,B 0,C 180,E1 8034.436,E2 8034.436} C_VEL
LIN {X 0,Y 147.426,Z 332.433,A -85,B 0,C 180,E1 8028.175,E2 8028.175} C_VEL
LIN {X 0,Y 147.423,Z 332.41,A -85,B 0,C 180,E1 8021.737,E2 8021.737} C_VEL
LIN {X 0,Y 147.428,Z 332.412,A -85,B 0,C 180,E1 8015.445,E2 8015.445} C_VEL
LIN {X 0,Y 147.435,Z 332.43,A -85,B 0,C 180,E1 8008.831,E2 8008.831} C_VEL
LIN {X 0,Y 147.43,Z 332.434,A -85,B 0,C 180,E1 8002.201,E2 8002.201} C_VEL
LIN {X 0,Y 147.432,Z 332.432,A -85,B 0,C 180,E1 7995.856,E2 7995.856} C_VEL
LIN {X 0,Y 147.452,Z 332.576,A -85,B 0,C 180,E1 7994.057,E2 7994.057} C_VEL
LIN {X 0,Y 150.278,Z 340.631,A -85,B 0,C 180,E1 7988.532,E2 7988.532} C_VEL
LIN {X 0,Y 153.062,Z 348.837,A -85,B 0,C 180,E1 7983.486,E2 7983.486} C_VEL
LIN {X 0,Y 156.166,Z 359.043,A -85,B 0,C 180,E1 7977.896,E2 7977.896} C_VEL
LIN {X 0,Y 159.366,Z 371.018,A -85,B 0,C 180,E1 7972.056,E2 7972.056} C_VEL
LIN {X 0,Y 162.516,Z 384.391,A -85,B 0,C 180,E1 7966.196,E2 7966.196} C_VEL
LIN {X 0,Y 164.809,Z 395.22,A -85,B 0,C 180,E1 7961.855,E2 7961.855} C_VEL
LIN {X 0,Y 163.645,Z 399.22,A -85,B 0,C 180,E1 7960.71,E2 7960.71} C_VEL
LIN {X 0,Y 163.765,Z 427.084,A -85,B 0,C 180,E1 7958.279,E2 7958.279} C_VEL
LIN {X 0,Y 164.748,Z 451.352,A -85,B 0,C 180,E1 7956.071,E2 7956.071} C_VEL
LIN {X 0,Y 155.909,Z 545.831,A -85,B 0,C 180,E1 7948.492,E2 7948.492} C_VEL
LIN {X 0,Y 154.033,Z 565.368,A -85,B 0,C 180,E1 7946.187,E2 7946.187} C_VEL
LIN {X 0,Y 151.965,Z 583.828,A -85,B 0,C 180,E1 7943.245,E2 7943.245} C_VEL
LIN {X 0,Y 149.964,Z 601.215,A -85,B 0,C 180,E1 7939.67,E2 7939.67} C_VEL
LIN {X 0,Y 148.139,Z 618.005,A -85,B 0,C 180,E1 7935.256,E2 7935.256} C_VEL
LIN {X 0,Y 146.907,Z 632.73,A -85,B 0,C 180,E1 7930.385,E2 7930.385} C_VEL
LIN {X 0,Y 146.416,Z 644.794,A -85,B 0,C 180,E1 7925.48,E2 7925.48} C_VEL
LIN {X 0,Y 146.717,Z 655.866,A -85,B 0,C 180,E1 7919.994,E2 7919.994} C_VEL
LIN {X 0,Y 148.005,Z 664.85,A -85,B 0,C 180,E1 7914.568,E2 7914.568} C_VEL
LIN {X 0,Y 151.139,Z 673.49,A -85,B 0,C 180,E1 7908.161,E2 7908.161} C_VEL
LIN {X 0,Y 155.794,Z 679.683,A -85,B 0,C 180,E1 7902.439,E2 7902.439} C_VEL
LIN {X 0,Y 162.536,Z 684.383,A -85,B 0,C 180,E1 7896.81,E2 7896.81} C_VEL
LIN {X 0,Y 171.545,Z 687.507,A -85,B 0,C 180,E1 7891.444,E2 7891.444} C_VEL
LIN {X 0,Y 182.235,Z 688.762,A -85,B 0,C 180,E1 7886.72,E2 7886.72} C_VEL
LIN {X 0,Y 194.173,Z 688.351,A -85,B 0,C 180,E1 7882.591,E2 7882.591} C_VEL
LIN {X 0,Y 178.696,Z 694.667,A -85,B 0,C 180,E1 7877.614,E2 7877.614} C_VEL
LIN {X 0,Y 165.284,Z 699.716,A -85,B 0,C 180,E1 7871.256,E2 7871.256} C_VEL
LIN {X 0,Y 155.14,Z 703.258,A -85,B 0,C 180,E1 7863.663,E2 7863.663} C_VEL
LIN {X 0,Y 148.719,Z 705.242,A -85,B 0,C 180,E1 7854.811,E2 7854.811} C_VEL
LIN {X 0,Y 146.729,Z 705.428,A -85,B 0,C 180,E1 7845.82,E2 7845.82} C_VEL
LIN {X 0,Y 148.269,Z 703.838,A -85,B 0,C 180,E1 7837.364,E2 7837.364} C_VEL
LIN {X 0,Y 150.726,Z 701.324,A -85,B 0,C 180,E1 7831.523,E2 7831.523} C_VEL
LIN {X 0,Y 150.971,Z 699.889,A -85,B 0,C 180,E1 7829.623,E2 7829.623} C_VEL
LIN {X 0,Y 149.902,Z 694.789,A -85,B 0,C 180,E1 7825.029,E2 7825.029} C_VEL
LIN {X 0,Y 148.938,Z 686.938,A -85,B 0,C 180,E1 7819.56,E2 7819.56} C_VEL
LIN {X 0,Y 148.753,Z 681.277,A -85,B 0,C 180,E1 7816.261,E2 7816.261} C_VEL
LIN {X 0,Y 147.88,Z 676.503,A -85,B 0,C 180,E1 7813.922,E2 7813.922} C_VEL
LIN {X 0,Y 144.492,Z 667.331,A -85,B 0,C 180,E1 7810.3,E2 7810.3} C_VEL
LIN {X 0,Y 142.757,Z 659.98,A -85,B 0,C 180,E1 7807.615,E2 7807.615} C_VEL
LIN {X 0,Y 142.831,Z 656.68,A -85,B 0,C 180,E1 7806.401,E2 7806.401} C_VEL
LIN {X 0,Y 145.137,Z 641.695,A -85,B 0,C 180,E1 7801.397,E2 7801.397} C_VEL
LIN {X 0,Y 147.887,Z 625.952,A -85,B 0,C 180,E1 7797.26,E2 7797.26} C_VEL
LIN {X 0,Y 150.974,Z 608.19,A -85,B 0,C 180,E1 7793.652,E2 7793.652} C_VEL
LIN {X 0,Y 153.825,Z 590.372,A -85,B 0,C 180,E1 7790.917,E2 7790.917} C_VEL
LIN {X 0,Y 156.124,Z 571.675,A -85,B 0,C 180,E1 7788.832,E2 7788.832} C_VEL
LIN {X 0,Y 159.941,Z 526.864,A -85,B 0,C 180,E1 7785.452,E2 7785.452} C_VEL
LIN {X 0,Y 169.264,Z 430.859,A -85,B 0,C 180,E1 7779.071,E2 7779.071} C_VEL
LIN {X 0,Y 168.825,Z 417.564,A -85,B 0,C 180,E1 7777.998,E2 7777.998} C_VEL
LIN {X 0,Y 158.899,Z 392.937,A -85,B 0,C 180,E1 7774.487,E2 7774.487} C_VEL
LIN {X 0,Y 154.469,Z 377.623,A -85,B 0,C 180,E1 7768.203,E2 7768.203} C_VEL
LIN {X 0,Y 150.822,Z 365.65,A -85,B 0,C 180,E1 7762.618,E2 7762.618} C_VEL
LIN {X 0,Y 147.33,Z 354.986,A -85,B 0,C 180,E1 7756.972,E2 7756.972} C_VEL
LIN {X 0,Y 144.19,Z 346.092,A -85,B 0,C 180,E1 7751.607,E2 7751.607} C_VEL
LIN {X 0,Y 141.546,Z 339.218,A -85,B 0,C 180,E1 7746.903,E2 7746.903} C_VEL
LIN {X 0,Y 140.255,Z 336.021,A -85,B 0,C 180,E1 7744.503,E2 7744.503} C_VEL
LIN {X 0,Y 139.464,Z 333.412,A -85,B 0,C 180,E1 7742.471,E2 7742.471} C_VEL
LIN {X 0,Y 139.468,Z 333.408,A -85,B 0,C 180,E1 7735.895,E2 7735.895} C_VEL
LIN {X 0,Y 139.469,Z 333.401,A -85,B 0,C 180,E1 7729.142,E2 7729.142} C_VEL
LIN {X 0,Y 139.473,Z 333.404,A -85,B 0,C 180,E1 7722.914,E2 7722.914} C_VEL
LIN {X 0,Y 139.476,Z 333.424,A -85,B 0,C 180,E1 7716.338,E2 7716.338} C_VEL
LIN {X 0,Y 139.491,Z 333.385,A -85,B 0,C 180,E1 7709.416,E2 7709.416} C_VEL
LIN {X 0,Y 139.476,Z 333.41,A -85,B 0,C 180,E1 7702.718,E2 7702.718} C_VEL
LIN {X 0,Y 139.475,Z 333.397,A -85,B 0,C 180,E1 7696.384,E2 7696.384} C_VEL
LIN {X 0,Y 139.488,Z 333.397,A -85,B 0,C 180,E1 7689.636,E2 7689.636} C_VEL
LIN {X 0,Y 139.486,Z 333.409,A -85,B 0,C 180,E1 7683.006,E2 7683.006} C_VEL
LIN {X 0,Y 139.482,Z 333.388,A -85,B 0,C 180,E1 7676.372,E2 7676.372} C_VEL
LIN {X 0,Y 139.49,Z 333.42,A -85,B 0,C 180,E1 7669.684,E2 7669.684} C_VEL
LIN {X 0,Y 139.487,Z 333.389,A -85,B 0,C 180,E1 7662.836,E2 7662.836} C_VEL
LIN {X 0,Y 139.485,Z 333.407,A -85,B 0,C 180,E1 7656.169,E2 7656.169} C_VEL
LIN {X 0,Y 139.499,Z 333.422,A -85,B 0,C 180,E1 7649.586,E2 7649.586} C_VEL
LIN {X 0,Y 139.495,Z 333.423,A -85,B 0,C 180,E1 7642.584,E2 7642.584} C_VEL
LIN {X 0,Y 139.528,Z 333.638,A -85,B 0,C 180,E1 7637.162,E2 7637.162} C_VEL
LIN {X 0,Y 142.203,Z 341.002,A -85,B 0,C 180,E1 7631.551,E2 7631.551} C_VEL
LIN {X 0,Y 145.048,Z 349.253,A -85,B 0,C 180,E1 7625.999,E2 7625.999} C_VEL
LIN {X 0,Y 147.943,Z 358.603,A -85,B 0,C 180,E1 7620.435,E2 7620.435} C_VEL
LIN {X 0,Y 151.059,Z 370.114,A -85,B 0,C 180,E1 7614.372,E2 7614.372} C_VEL
LIN {X 0,Y 154.021,Z 382.511,A -85,B 0,C 180,E1 7608.532,E2 7608.532} C_VEL
LIN {X 0,Y 156.984,Z 396.406,A -85,B 0,C 180,E1 7602.608,E2 7602.608} C_VEL
LIN {X 0,Y 156.269,Z 399.097,A -85,B 0,C 180,E1 7601.83,E2 7601.83} C_VEL
LIN {X 0,Y 156.189,Z 425.85,A -85,B 0,C 180,E1 7599.402,E2 7599.402} C_VEL
LIN {X 0,Y 157.104,Z 451.677,A -85,B 0,C 180,E1 7596.936,E2 7596.936} C_VEL
LIN {X 0,Y 147.975,Z 546.111,A -85,B 0,C 180,E1 7588.938,E2 7588.938} C_VEL
LIN {X 0,Y 146.126,Z 564.952,A -85,B 0,C 180,E1 7586.62,E2 7586.62} C_VEL
LIN {X 0,Y 143.997,Z 583.574,A -85,B 0,C 180,E1 7583.525,E2 7583.525} C_VEL
LIN {X 0,Y 141.852,Z 601.903,A -85,B 0,C 180,E1 7579.554,E2 7579.554} C_VEL
LIN {X 0,Y 140.037,Z 618.664,A -85,B 0,C 180,E1 7574.888,E2 7574.888} C_VEL
LIN {X 0,Y 138.893,Z 632.852,A -85,B 0,C 180,E1 7569.943,E2 7569.943} C_VEL
LIN {X 0,Y 138.468,Z 645.038,A -85,B 0,C 180,E1 7564.775,E2 7564.775} C_VEL
LIN {X 0,Y 138.946,Z 656.592,A -85,B 0,C 180,E1 7558.757,E2 7558.757} C_VEL
LIN {X 0,Y 140.659,Z 666.249,A -85,B 0,C 180,E1 7552.643,E2 7552.643} C_VEL
LIN {X 0,Y 144.371,Z 674.873,A -85,B 0,C 180,E1 7545.966,E2 7545.966} C_VEL
LIN {X 0,Y 150.058,Z 681.458,A -85,B 0,C 180,E1 7539.722,E2 7539.722} C_VEL
LIN {X 0,Y 158.149,Z 686.384,A -85,B 0,C 180,E1 7533.728,E2 7533.728} C_VEL
LIN {X 0,Y 168.146,Z 689.472,A -85,B 0,C 180,E1 7528.442,E2 7528.442} C_VEL
LIN {X 0,Y 179.767,Z 690.735,A -85,B 0,C 180,E1 7523.869,E2 7523.869} C_VEL
LIN {X 0,Y 182.946,Z 690.827,A -85,B 0,C 180,E1 7522.748,E2 7522.748} C_VEL
LIN {X 0,Y 167.509,Z 696.031,A -85,B 0,C 180,E1 7517.242,E2 7517.242} C_VEL
LIN {X 0,Y 154.528,Z 699.954,A -85,B 0,C 180,E1 7510.219,E2 7510.219} C_VEL
LIN {X 0,Y 144.981,Z 702.434,A -85,B 0,C 180,E1 7501.613,E2 7501.613} C_VEL
LIN {X 0,Y 139.991,Z 703.246,A -85,B 0,C 180,E1 7492.247,E2 7492.247} C_VEL
LIN {X 0,Y 139.414,Z 702.336,A -85,B 0,C 180,E1 7482.72,E2 7482.72} C_VEL
LIN {X 0,Y 141.952,Z 699.835,A -85,B 0,C 180,E1 7474.447,E2 7474.447} C_VEL
LIN {X 0,Y 143.553,Z 697.894,A -85,B 0,C 180,E1 7470.801,E2 7470.801} C_VEL
LIN {X 0,Y 142.715,Z 693.778,A -85,B 0,C 180,E1 7466.79,E2 7466.79} C_VEL
LIN {X 0,Y 141.51,Z 686.152,A -85,B 0,C 180,E1 7461.061,E2 7461.061} C_VEL
LIN {X 0,Y 141.154,Z 676.38,A -85,B 0,C 180,E1 7455.229,E2 7455.229} C_VEL
LIN {X 0,Y 141.881,Z 664.698,A -85,B 0,C 180,E1 7449.612,E2 7449.612} C_VEL
LIN {X 0,Y 142.831,Z 656.68,A -85,B 0,C 180,E1 7446.401,E2 7446.401} C_VEL
LIN {X 0,Y 142.673,Z 650.83,A -85,B 0,C 180,E1 7444.394,E2 7444.394} C_VEL
LIN {X 0,Y 140.241,Z 640.143,A -85,B 0,C 180,E1 7441.252,E2 7441.252} C_VEL
LIN {X 0,Y 139.099,Z 631.742,A -85,B 0,C 180,E1 7438.997,E2 7438.997} C_VEL
LIN {X 0,Y 139.41,Z 627.91,A -85,B 0,C 180,E1 7438,E2 7438} C_VEL
LIN {X 0,Y 142.261,Z 611.839,A -85,B 0,C 180,E1 7434.317,E2 7434.317} C_VEL
LIN {X 0,Y 145.224,Z 593.971,A -85,B 0,C 180,E1 7431.21,E2 7431.21} C_VEL
LIN {X 0,Y 147.774,Z 575.545,A -85,B 0,C 180,E1 7428.826,E2 7428.826} C_VEL
LIN {X 0,Y 149.858,Z 552.587,A -85,B 0,C 180,E1 7426.791,E2 7426.791} C_VEL
LIN {X 0,Y 161.778,Z 431.15,A -85,B 0,C 180,E1 7418.08,E2 7418.08} C_VEL
LIN {X 0,Y 161.385,Z 419.767,A -85,B 0,C 180,E1 7417.111,E2 7417.111} C_VEL
